KUKA KRL program: EPS_2_25716_MHDR06_A_20250926071555.src

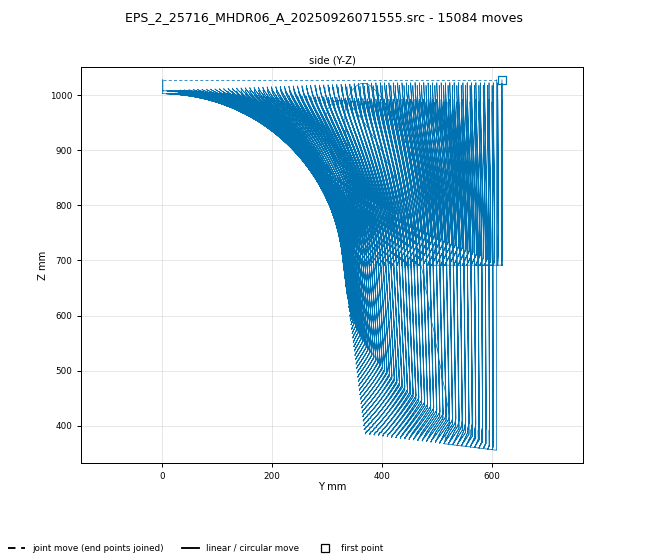
[picture p0: tool path of EPS_2_25716_MHDR06_A_20250926071555.src, 15084 of 15086 moves have a stored position in this frame; points joined in program order, loops and branches not executed]
&ACCESS RVP
&REL 4
&COMMENT QRS 19112012
&PARAM EDITMASK = *
DEF PART()
EXT BAS (BAS_COMMAND :IN,REAL :IN )
INT I
BAS (#INITMOV,0 )

;KUKA QRS Post kuka4.cps  Date:22-06-2017 !

File_ID=2855

QRS_PRE_INIT()

;Init var - Until changes are made in qrs_pre_init
Outlet_Square_prg=0
Inlet_1_Square_prg=0
Inlet_2_Square_prg=0
Inlet_3_Square_prg=0
Inlet_4_Square_prg=0
Inlet_5_Square_prg=0

Outlet_1={X 0.000, Y 400.000, Z 713.000, B 0.000, E1 0.000 }
Inlet_1={X 0.000, Y 400.000, Z 683.000, B 0.000, E1 180.000 }
Outlet_1_type=610
Inlet_1_type=610
;QRS#1=Sidecore dimensions
;QRS#2=600-24" Concrete
;QRS#3=600-24" Concrete
;QRS#4=
;QRS#5=
;QRS#6=
;QRS#7=
;QRS#8=
;QRS#9=S306-34L
;QRS#10=S306-34L
;QRS#11=
;QRS#12=
;QRS#13=
;QRS#14=
;QRS#15=
;QRS#16=1220x127x1372 4,5'
;QRS#17=EPS Height
;QRS#18=1018
;QRS#19=*
;QRS#20= UPDATED VERSION 22-06-2017
;QRS#21=*
Outlet_Square=0450
Inlet_1_Square=0450
Inlet_2_Square=0
Inlet_3_Square=0
Inlet_4_Square=0
Inlet_5_Square=0
Mill_Square=1
Outlet_Square_Prg=264
Inlet_1_Square_prg=264

QRS_INIT()

$ADVANCE=5

; T1
PTP {E1 171.02,E2 171.02}
PTP {X 0,Y 617.769,A -85,B 0,C 180,E1 171.02,E2 171.02,E3 0,E4 0,E5 0,E6 0}
QRS_SPEED_INIT()
LIN {X 0,Y 617.769,Z 1028,A -85,B 0,C 180,E1 171.02,E2 171.02,E3 0,E4 0,E5 0,E6 0} C_VEL
LIN {X 0,Y 617.769,Z 693.44,A -85,B 0,C 180,E1 171.02,E2 171.02} C_VEL
LIN {X 0,Y 617.8,Z 691.44,A -85,B 0,C 180,E1 171.206,E2 171.206} C_VEL
LIN {X 0,Y 617.968,Z 691.44,A -85,B 0,C 180,E1 171.885,E2 171.885} C_VEL
LIN {X 0,Y 618.013,Z 691.44,A -85,B 0,C 180,E1 176.532,E2 176.532} C_VEL
LIN {X 0,Y 618.047,Z 691.44,A -85,B 0,C 180,E1 181.155,E2 181.155} C_VEL
LIN {X 0,Y 617.982,Z 691.44,A -85,B 0,C 180,E1 185.787,E2 185.787} C_VEL
LIN {X 0,Y 617.952,Z 691.44,A -85,B 0,C 180,E1 190.457,E2 190.457} C_VEL
LIN {X 0,Y 617.972,Z 691.44,A -85,B 0,C 180,E1 195.197,E2 195.197} C_VEL
LIN {X 0,Y 617.907,Z 691.44,A -85,B 0,C 180,E1 200.05,E2 200.05} C_VEL
LIN {X 0,Y 617.438,Z 691.44,A -85,B 0,C 180,E1 202.548,E2 202.548} C_VEL
LIN {X 0,Y 617.908,Z 691.44,A -85,B 0,C 180,E1 205.056,E2 205.056} C_VEL
LIN {X 0,Y 617.398,Z 691.44,A -85,B 0,C 180,E1 207.66,E2 207.66} C_VEL
LIN {X 0,Y 617.843,Z 691.44,A -85,B 0,C 180,E1 210.28,E2 210.28} C_VEL
LIN {X 0,Y 617.317,Z 691.44,A -85,B 0,C 180,E1 213.027,E2 213.027} C_VEL
LIN {X 0,Y 617.82,Z 691.44,A -85,B 0,C 180,E1 215.798,E2 215.798} C_VEL
LIN {X 0,Y 617.574,Z 691.44,A -85,B 0,C 180,E1 218.108,E2 218.108} C_VEL
LIN {X 0,Y 617.547,Z 691.44,A -85,B 0,C 180,E1 218.722,E2 218.722} C_VEL
LIN {X 0,Y 617.751,Z 691.44,A -85,B 0,C 180,E1 221.735,E2 221.735} C_VEL
LIN {X 0,Y 617.856,Z 691.44,A -85,B 0,C 180,E1 225.104,E2 225.104} C_VEL
LIN {X 0,Y 617.438,Z 691.44,A -85,B 0,C 180,E1 228.31,E2 228.31} C_VEL
LIN {X 0,Y 617.785,Z 691.44,A -85,B 0,C 180,E1 231.301,E2 231.301} C_VEL
LIN {X 0,Y 617.972,Z 691.44,A -85,B 0,C 180,E1 236.345,E2 236.345} C_VEL
LIN {X 0,Y 617.889,Z 691.44,A -85,B 0,C 180,E1 236.677,E2 236.677} C_VEL
LIN {X 0,Y 617.182,Z 691.44,A -85,B 0,C 180,E1 236.802,E2 236.802} C_VEL
LIN {X 0,Y 616.593,Z 691.442,A -85,B 0,C 180,E1 236.859,E2 236.859} C_VEL
LIN {X 0,Y 617.379,Z 698.721,A -85,B 0,C 180,E1 237.005,E2 237.005} C_VEL
LIN {X 0,Y 617.562,Z 731.83,A -85,B 0,C 180,E1 237.472,E2 237.472} C_VEL
LIN {X 0,Y 617.518,Z 745.273,A -85,B 0,C 180,E1 237.692,E2 237.692} C_VEL
LIN {X 0,Y 617.627,Z 759.991,A -85,B 0,C 180,E1 238.015,E2 238.015} C_VEL
LIN {X 0,Y 617.596,Z 772.178,A -85,B 0,C 180,E1 238.333,E2 238.333} C_VEL
LIN {X 0,Y 617.775,Z 789.25,A -85,B 0,C 180,E1 238.876,E2 238.876} C_VEL
LIN {X 0,Y 617.661,Z 803.567,A -85,B 0,C 180,E1 239.398,E2 239.398} C_VEL
LIN {X 0,Y 617.795,Z 819.272,A -85,B 0,C 180,E1 240.077,E2 240.077} C_VEL
LIN {X 0,Y 617.796,Z 833.607,A -85,B 0,C 180,E1 240.772,E2 240.772} C_VEL
LIN {X 0,Y 617.742,Z 845.603,A -85,B 0,C 180,E1 241.41,E2 241.41} C_VEL
LIN {X 0,Y 617.842,Z 859.517,A -85,B 0,C 180,E1 242.243,E2 242.243} C_VEL
LIN {X 0,Y 617.838,Z 873.674,A -85,B 0,C 180,E1 243.177,E2 243.177} C_VEL
LIN {X 0,Y 617.828,Z 885.936,A -85,B 0,C 180,E1 244.063,E2 244.063} C_VEL
LIN {X 0,Y 617.821,Z 897.15,A -85,B 0,C 180,E1 244.943,E2 244.943} C_VEL
LIN {X 0,Y 617.854,Z 908.216,A -85,B 0,C 180,E1 245.886,E2 245.886} C_VEL
LIN {X 0,Y 617.903,Z 919.181,A -85,B 0,C 180,E1 246.901,E2 246.901} C_VEL
LIN {X 0,Y 617.832,Z 929.557,A -85,B 0,C 180,E1 247.938,E2 247.938} C_VEL
LIN {X 0,Y 617.851,Z 939.544,A -85,B 0,C 180,E1 249.026,E2 249.026} C_VEL
LIN {X 0,Y 617.957,Z 948.912,A -85,B 0,C 180,E1 250.137,E2 250.137} C_VEL
LIN {X 0,Y 617.805,Z 957.463,A -85,B 0,C 180,E1 251.226,E2 251.226} C_VEL
LIN {X 0,Y 617.797,Z 965.811,A -85,B 0,C 180,E1 252.391,E2 252.391} C_VEL
LIN {X 0,Y 617.997,Z 973.741,A -85,B 0,C 180,E1 253.613,E2 253.613} C_VEL
LIN {X 0,Y 617.808,Z 980.894,A -85,B 0,C 180,E1 254.801,E2 254.801} C_VEL
LIN {X 0,Y 617.811,Z 988.821,A -85,B 0,C 180,E1 256.292,E2 256.292} C_VEL
LIN {X 0,Y 617.963,Z 994.484,A -85,B 0,C 180,E1 257.482,E2 257.482} C_VEL
LIN {X 0,Y 617.732,Z 1000.738,A -85,B 0,C 180,E1 258.953,E2 258.953} C_VEL
LIN {X 0,Y 617.807,Z 1005.633,A -85,B 0,C 180,E1 260.289,E2 260.289} C_VEL
LIN {X 0,Y 617.976,Z 1008.324,A -85,B 0,C 180,E1 261.143,E2 261.143} C_VEL
LIN {X 0,Y 617.856,Z 1010.563,A -85,B 0,C 180,E1 261.885,E2 261.885} C_VEL
LIN {X 0,Y 617.743,Z 1013.111,A -85,B 0,C 180,E1 262.816,E2 262.816} C_VEL
LIN {X 0,Y 617.83,Z 1016.208,A -85,B 0,C 180,E1 264.213,E2 264.213} C_VEL
LIN {X 0,Y 617.976,Z 1017.804,A -85,B 0,C 180,E1 265.143,E2 265.143} C_VEL
LIN {X 0,Y 617.882,Z 1018.62,A -85,B 0,C 180,E1 265.605,E2 265.605} C_VEL
LIN {X 0,Y 617.751,Z 1019.844,A -85,B 0,C 180,E1 266.531,E2 266.531} C_VEL
LIN {X 0,Y 617.754,Z 1020.831,A -85,B 0,C 180,E1 267.457,E2 267.457} C_VEL
LIN {X 0,Y 617.996,Z 1021.643,A -85,B 0,C 180,E1 268.845,E2 268.845} C_VEL
LIN {X 0,Y 617.666,Z 1021.732,A -85,B 0,C 180,E1 271.156,E2 271.156} C_VEL
LIN {X 0,Y 617.88,Z 1020.797,A -85,B 0,C 180,E1 272.543,E2 272.543} C_VEL
LIN {X 0,Y 617.842,Z 1019.819,A -85,B 0,C 180,E1 273.469,E2 273.469} C_VEL
LIN {X 0,Y 617.732,Z 1018.658,A -85,B 0,C 180,E1 274.396,E2 274.396} C_VEL
LIN {X 0,Y 617.804,Z 1016.213,A -85,B 0,C 180,E1 275.788,E2 275.788} C_VEL
LIN {X 0,Y 617.988,Z 1014.126,A -85,B 0,C 180,E1 276.716,E2 276.716} C_VEL
LIN {X 0,Y 617.83,Z 1011.822,A -85,B 0,C 180,E1 277.649,E2 277.649} C_VEL
LIN {X 0,Y 617.78,Z 1008.462,A -85,B 0,C 180,E1 278.832,E2 278.832} C_VEL
LIN {X 0,Y 617.963,Z 1004.405,A -85,B 0,C 180,E1 280.048,E2 280.048} C_VEL
LIN {X 0,Y 617.795,Z 999.566,A -85,B 0,C 180,E1 281.341,E2 281.341} C_VEL
LIN {X 0,Y 617.74,Z 994.527,A -85,B 0,C 180,E1 282.523,E2 282.523} C_VEL
LIN {X 0,Y 617.975,Z 987.305,A -85,B 0,C 180,E1 284.002,E2 284.002} C_VEL
LIN {X 0,Y 617.805,Z 979.862,A -85,B 0,C 180,E1 285.374,E2 285.374} C_VEL
LIN {X 0,Y 617.795,Z 972.028,A -85,B 0,C 180,E1 286.666,E2 286.666} C_VEL
LIN {X 0,Y 617.958,Z 964.032,A -85,B 0,C 180,E1 287.857,E2 287.857} C_VEL
LIN {X 0,Y 617.819,Z 955.95,A -85,B 0,C 180,E1 288.977,E2 288.977} C_VEL
LIN {X 0,Y 617.839,Z 946.158,A -85,B 0,C 180,E1 290.204,E2 290.204} C_VEL
LIN {X 0,Y 617.952,Z 936.782,A -85,B 0,C 180,E1 291.281,E2 291.281} C_VEL
LIN {X 0,Y 617.847,Z 926.511,A -85,B 0,C 180,E1 292.374,E2 292.374} C_VEL
LIN {X 0,Y 617.845,Z 916.724,A -85,B 0,C 180,E1 293.335,E2 293.335} C_VEL
LIN {X 0,Y 617.862,Z 905.186,A -85,B 0,C 180,E1 294.376,E2 294.376} C_VEL
LIN {X 0,Y 617.853,Z 894.173,A -85,B 0,C 180,E1 295.295,E2 295.295} C_VEL
LIN {X 0,Y 617.838,Z 881.592,A -85,B 0,C 180,E1 296.259,E2 296.259} C_VEL
LIN {X 0,Y 617.824,Z 870.134,A -85,B 0,C 180,E1 297.067,E2 297.067} C_VEL
LIN {X 0,Y 617.85,Z 856.712,A -85,B 0,C 180,E1 297.928,E2 297.928} C_VEL
LIN {X 0,Y 617.812,Z 842.841,A -85,B 0,C 180,E1 298.735,E2 298.735} C_VEL
LIN {X 0,Y 617.728,Z 831.67,A -85,B 0,C 180,E1 299.334,E2 299.334} C_VEL
LIN {X 0,Y 617.799,Z 815.203,A -85,B 0,C 180,E1 300.103,E2 300.103} C_VEL
LIN {X 0,Y 617.676,Z 801.179,A -85,B 0,C 180,E1 300.691,E2 300.691} C_VEL
LIN {X 0,Y 617.671,Z 792.906,A -85,B 0,C 180,E1 300.996,E2 300.996} C_VEL
LIN {X 0,Y 617.767,Z 783.913,A -85,B 0,C 180,E1 301.296,E2 301.296} C_VEL
LIN {X 0,Y 617.782,Z 774.18,A -85,B 0,C 180,E1 301.602,E2 301.602} C_VEL
LIN {X 0,Y 617.522,Z 758.624,A -85,B 0,C 180,E1 302.025,E2 302.025} C_VEL
LIN {X 0,Y 617.763,Z 743.298,A -85,B 0,C 180,E1 302.332,E2 302.332} C_VEL
LIN {X 0,Y 617.696,Z 723.174,A -85,B 0,C 180,E1 302.644,E2 302.644} C_VEL
LIN {X 0,Y 617.36,Z 698.518,A -85,B 0,C 180,E1 302.998,E2 302.998} C_VEL
LIN {X 0,Y 616.602,Z 691.44,A -85,B 0,C 180,E1 303.143,E2 303.143} C_VEL
LIN {X 0,Y 617.104,Z 691.44,A -85,B 0,C 180,E1 303.189,E2 303.189} C_VEL
LIN {X 0,Y 617.789,Z 691.44,A -85,B 0,C 180,E1 303.3,E2 303.3} C_VEL
LIN {X 0,Y 618.014,Z 691.44,A -85,B 0,C 180,E1 303.592,E2 303.592} C_VEL
LIN {X 0,Y 617.789,Z 691.44,A -85,B 0,C 180,E1 308.699,E2 308.699} C_VEL
LIN {X 0,Y 617.439,Z 691.44,A -85,B 0,C 180,E1 311.755,E2 311.755} C_VEL
LIN {X 0,Y 617.857,Z 691.44,A -85,B 0,C 180,E1 314.897,E2 314.897} C_VEL
LIN {X 0,Y 617.756,Z 691.44,A -85,B 0,C 180,E1 318.27,E2 318.27} C_VEL
LIN {X 0,Y 617.543,Z 691.44,A -85,B 0,C 180,E1 321.278,E2 321.278} C_VEL
LIN {X 0,Y 617.577,Z 691.44,A -85,B 0,C 180,E1 321.893,E2 321.893} C_VEL
LIN {X 0,Y 617.818,Z 691.44,A -85,B 0,C 180,E1 324.202,E2 324.202} C_VEL
LIN {X 0,Y 617.322,Z 691.44,A -85,B 0,C 180,E1 326.974,E2 326.974} C_VEL
LIN {X 0,Y 617.835,Z 691.44,A -85,B 0,C 180,E1 329.719,E2 329.719} C_VEL
LIN {X 0,Y 617.381,Z 691.44,A -85,B 0,C 180,E1 332.339,E2 332.339} C_VEL
LIN {X 0,Y 617.882,Z 691.44,A -85,B 0,C 180,E1 334.943,E2 334.943} C_VEL
LIN {X 0,Y 617.416,Z 691.44,A -85,B 0,C 180,E1 337.451,E2 337.451} C_VEL
LIN {X 0,Y 617.909,Z 691.44,A -85,B 0,C 180,E1 339.95,E2 339.95} C_VEL
LIN {X 0,Y 617.993,Z 691.44,A -85,B 0,C 180,E1 343.627,E2 343.627} C_VEL
LIN {X 0,Y 617.927,Z 691.44,A -85,B 0,C 180,E1 349.543,E2 349.543} C_VEL
LIN {X 0,Y 617.984,Z 691.44,A -85,B 0,C 180,E1 354.213,E2 354.213} C_VEL
LIN {X 0,Y 618.053,Z 691.44,A -85,B 0,C 180,E1 358.845,E2 358.845} C_VEL
LIN {X 0,Y 618.006,Z 691.44,A -85,B 0,C 180,E1 363.468,E2 363.468} C_VEL
LIN {X 0,Y 617.974,Z 691.44,A -85,B 0,C 180,E1 368.115,E2 368.115} C_VEL
LIN {X 0,Y 617.996,Z 691.44,A -85,B 0,C 180,E1 372.815,E2 372.815} C_VEL
LIN {X 0,Y 617.957,Z 691.44,A -85,B 0,C 180,E1 377.607,E2 377.607} C_VEL
LIN {X 0,Y 617.756,Z 691.44,A -85,B 0,C 180,E1 378.561,E2 378.561} C_VEL
LIN {X 0,Y 617.91,Z 691.44,A -85,B 0,C 180,E1 382.53,E2 382.53} C_VEL
LIN {X 0,Y 617.424,Z 691.44,A -85,B 0,C 180,E1 385.077,E2 385.077} C_VEL
LIN {X 0,Y 617.883,Z 691.44,A -85,B 0,C 180,E1 387.637,E2 387.637} C_VEL
LIN {X 0,Y 617.432,Z 691.44,A -85,B 0,C 180,E1 390.302,E2 390.302} C_VEL
LIN {X 0,Y 617.966,Z 691.44,A -85,B 0,C 180,E1 392.988,E2 392.988} C_VEL
LIN {X 0,Y 617.693,Z 691.44,A -85,B 0,C 180,E1 395.806,E2 395.806} C_VEL
LIN {X 0,Y 617.694,Z 691.44,A -85,B 0,C 180,E1 398.121,E2 398.121} C_VEL
LIN {X 0,Y 617.812,Z 691.44,A -85,B 0,C 180,E1 401.736,E2 401.736} C_VEL
LIN {X 0,Y 617.415,Z 691.44,A -85,B 0,C 180,E1 405.062,E2 405.062} C_VEL
LIN {X 0,Y 617.817,Z 691.44,A -85,B 0,C 180,E1 408.276,E2 408.276} C_VEL
LIN {X 0,Y 617.727,Z 691.44,A -85,B 0,C 180,E1 411.882,E2 411.882} C_VEL
LIN {X 0,Y 617.729,Z 691.44,A -85,B 0,C 180,E1 414.2,E2 414.2} C_VEL
LIN {X 0,Y 617.795,Z 691.44,A -85,B 0,C 180,E1 415.792,E2 415.792} C_VEL
LIN {X 0,Y 617.754,Z 691.44,A -85,B 0,C 180,E1 417.003,E2 417.003} C_VEL
LIN {X 0,Y 617.547,Z 700.565,A -85,B 0,C 180,E1 417.406,E2 417.406} C_VEL
LIN {X 0,Y 617.667,Z 715.154,A -85,B 0,C 180,E1 417.653,E2 417.653} C_VEL
LIN {X 0,Y 617.521,Z 730.803,A -85,B 0,C 180,E1 417.985,E2 417.985} C_VEL
LIN {X 0,Y 617.762,Z 746.117,A -85,B 0,C 180,E1 418.413,E2 418.413} C_VEL
LIN {X 0,Y 617.721,Z 761.16,A -85,B 0,C 180,E1 418.898,E2 418.898} C_VEL
LIN {X 0,Y 617.647,Z 771.287,A -85,B 0,C 180,E1 419.267,E2 419.267} C_VEL
LIN {X 0,Y 617.812,Z 788.844,A -85,B 0,C 180,E1 420.012,E2 420.012} C_VEL
LIN {X 0,Y 617.71,Z 803.562,A -85,B 0,C 180,E1 420.72,E2 420.72} C_VEL
LIN {X 0,Y 617.82,Z 816.37,A -85,B 0,C 180,E1 421.414,E2 421.414} C_VEL
LIN {X 0,Y 617.848,Z 830.932,A -85,B 0,C 180,E1 422.29,E2 422.29} C_VEL
LIN {X 0,Y 617.783,Z 843.16,A -85,B 0,C 180,E1 423.093,E2 423.093} C_VEL
LIN {X 0,Y 617.824,Z 855.473,A -85,B 0,C 180,E1 423.982,E2 423.982} C_VEL
LIN {X 0,Y 617.846,Z 867.672,A -85,B 0,C 180,E1 424.944,E2 424.944} C_VEL
LIN {X 0,Y 617.863,Z 878.611,A -85,B 0,C 180,E1 425.878,E2 425.878} C_VEL
LIN {X 0,Y 617.83,Z 889.973,A -85,B 0,C 180,E1 426.932,E2 426.932} C_VEL
LIN {X 0,Y 617.877,Z 899.967,A -85,B 0,C 180,E1 427.939,E2 427.939} C_VEL
LIN {X 0,Y 617.955,Z 908.593,A -85,B 0,C 180,E1 428.874,E2 428.874} C_VEL
LIN {X 0,Y 617.815,Z 919.245,A -85,B 0,C 180,E1 430.128,E2 430.128} C_VEL
LIN {X 0,Y 617.837,Z 927.602,A -85,B 0,C 180,E1 431.202,E2 431.202} C_VEL
LIN {X 0,Y 617.942,Z 936.082,A -85,B 0,C 180,E1 432.394,E2 432.394} C_VEL
LIN {X 0,Y 617.763,Z 944.459,A -85,B 0,C 180,E1 433.676,E2 433.676} C_VEL
LIN {X 0,Y 617.824,Z 951.132,A -85,B 0,C 180,E1 434.8,E2 434.8} C_VEL
LIN {X 0,Y 617.979,Z 957.548,A -85,B 0,C 180,E1 435.998,E2 435.998} C_VEL
LIN {X 0,Y 617.736,Z 964.719,A -85,B 0,C 180,E1 437.477,E2 437.477} C_VEL
LIN {X 0,Y 617.804,Z 969.758,A -85,B 0,C 180,E1 438.659,E2 438.659} C_VEL
LIN {X 0,Y 617.968,Z 974.595,A -85,B 0,C 180,E1 439.958,E2 439.958} C_VEL
LIN {X 0,Y 617.756,Z 978.96,A -85,B 0,C 180,E1 441.275,E2 441.275} C_VEL
LIN {X 0,Y 617.845,Z 983.206,A -85,B 0,C 180,E1 442.817,E2 442.817} C_VEL
LIN {X 0,Y 617.962,Z 985.246,A -85,B 0,C 180,E1 443.749,E2 443.749} C_VEL
LIN {X 0,Y 617.792,Z 987.146,A -85,B 0,C 180,E1 444.676,E2 444.676} C_VEL
LIN {X 0,Y 617.736,Z 988.734,A -85,B 0,C 180,E1 445.604,E2 445.604} C_VEL
LIN {X 0,Y 617.822,Z 989.878,A -85,B 0,C 180,E1 446.531,E2 446.531} C_VEL
LIN {X 0,Y 617.972,Z 990.803,A -85,B 0,C 180,E1 447.457,E2 447.457} C_VEL
LIN {X 0,Y 617.716,Z 991.728,A -85,B 0,C 180,E1 448.844,E2 448.844} C_VEL
LIN {X 0,Y 617.923,Z 991.653,A -85,B 0,C 180,E1 451.155,E2 451.155} C_VEL
LIN {X 0,Y 617.765,Z 990.797,A -85,B 0,C 180,E1 452.543,E2 452.543} C_VEL
LIN {X 0,Y 617.677,Z 989.809,A -85,B 0,C 180,E1 453.469,E2 453.469} C_VEL
LIN {X 0,Y 617.742,Z 988.579,A -85,B 0,C 180,E1 454.396,E2 454.396} C_VEL
LIN {X 0,Y 617.919,Z 986.085,A -85,B 0,C 180,E1 455.786,E2 455.786} C_VEL
LIN {X 0,Y 617.727,Z 982.992,A -85,B 0,C 180,E1 457.184,E2 457.184} C_VEL
LIN {X 0,Y 617.798,Z 979.363,A -85,B 0,C 180,E1 458.507,E2 458.507} C_VEL
LIN {X 0,Y 617.934,Z 975.572,A -85,B 0,C 180,E1 459.674,E2 459.674} C_VEL
LIN {X 0,Y 617.754,Z 969.384,A -85,B 0,C 180,E1 461.341,E2 461.341} C_VEL
LIN {X 0,Y 617.889,Z 964.306,A -85,B 0,C 180,E1 462.52,E2 462.52} C_VEL
LIN {X 0,Y 617.89,Z 960.018,A -85,B 0,C 180,E1 463.409,E2 463.409} C_VEL
LIN {X 0,Y 617.758,Z 955.491,A -85,B 0,C 180,E1 464.304,E2 464.304} C_VEL
LIN {X 0,Y 617.765,Z 949.526,A -85,B 0,C 180,E1 465.387,E2 465.387} C_VEL
LIN {X 0,Y 617.977,Z 942.352,A -85,B 0,C 180,E1 466.563,E2 466.563} C_VEL
LIN {X 0,Y 617.805,Z 933.783,A -85,B 0,C 180,E1 467.854,E2 467.854} C_VEL
LIN {X 0,Y 617.794,Z 925.779,A -85,B 0,C 180,E1 468.954,E2 468.954} C_VEL
LIN {X 0,Y 617.962,Z 915.769,A -85,B 0,C 180,E1 470.199,E2 470.199} C_VEL
LIN {X 0,Y 617.846,Z 906.373,A -85,B 0,C 180,E1 471.284,E2 471.284} C_VEL
LIN {X 0,Y 617.826,Z 896.063,A -85,B 0,C 180,E1 472.374,E2 472.374} C_VEL
LIN {X 0,Y 617.902,Z 886.089,A -85,B 0,C 180,E1 473.345,E2 473.345} C_VEL
LIN {X 0,Y 617.877,Z 876.237,A -85,B 0,C 180,E1 474.242,E2 474.242} C_VEL
LIN {X 0,Y 617.845,Z 863.602,A -85,B 0,C 180,E1 475.295,E2 475.295} C_VEL
LIN {X 0,Y 617.816,Z 852.103,A -85,B 0,C 180,E1 476.178,E2 476.178} C_VEL
LIN {X 0,Y 617.858,Z 839.452,A -85,B 0,C 180,E1 477.065,E2 477.065} C_VEL
LIN {X 0,Y 617.837,Z 826.763,A -85,B 0,C 180,E1 477.88,E2 477.88} C_VEL
LIN {X 0,Y 617.724,Z 813.694,A -85,B 0,C 180,E1 478.649,E2 478.649} C_VEL
LIN {X 0,Y 617.815,Z 799.775,A -85,B 0,C 180,E1 479.376,E2 479.376} C_VEL
LIN {X 0,Y 617.769,Z 785.259,A -85,B 0,C 180,E1 480.058,E2 480.058} C_VEL
LIN {X 0,Y 617.652,Z 771.869,A -85,B 0,C 180,E1 480.622,E2 480.622} C_VEL
LIN {X 0,Y 617.768,Z 756.723,A -85,B 0,C 180,E1 481.162,E2 481.162} C_VEL
LIN {X 0,Y 617.634,Z 741.567,A -85,B 0,C 180,E1 481.635,E2 481.635} C_VEL
LIN {X 0,Y 617.622,Z 734.394,A -85,B 0,C 180,E1 481.825,E2 481.825} C_VEL
LIN {X 0,Y 617.755,Z 725.284,A -85,B 0,C 180,E1 482.038,E2 482.038} C_VEL
LIN {X 0,Y 617.77,Z 711.173,A -85,B 0,C 180,E1 482.321,E2 482.321} C_VEL
LIN {X 0,Y 617.397,Z 692.323,A -85,B 0,C 180,E1 482.628,E2 482.628} C_VEL
LIN {X 0,Y 617.467,Z 691.44,A -85,B 0,C 180,E1 482.656,E2 482.656} C_VEL
LIN {X 0,Y 618.076,Z 691.44,A -85,B 0,C 180,E1 482.977,E2 482.977} C_VEL
LIN {X 0,Y 617.727,Z 691.44,A -85,B 0,C 180,E1 484.199,E2 484.199} C_VEL
LIN {X 0,Y 617.784,Z 691.44,A -85,B 0,C 180,E1 488.699,E2 488.699} C_VEL
LIN {X 0,Y 617.435,Z 691.44,A -85,B 0,C 180,E1 491.755,E2 491.755} C_VEL
LIN {X 0,Y 617.864,Z 691.44,A -85,B 0,C 180,E1 494.895,E2 494.895} C_VEL
LIN {X 0,Y 617.761,Z 691.44,A -85,B 0,C 180,E1 498.268,E2 498.268} C_VEL
LIN {X 0,Y 617.553,Z 691.44,A -85,B 0,C 180,E1 501.278,E2 501.278} C_VEL
LIN {X 0,Y 617.828,Z 691.44,A -85,B 0,C 180,E1 504.203,E2 504.203} C_VEL
LIN {X 0,Y 617.326,Z 691.44,A -85,B 0,C 180,E1 506.974,E2 506.974} C_VEL
LIN {X 0,Y 617.855,Z 691.44,A -85,B 0,C 180,E1 509.72,E2 509.72} C_VEL
LIN {X 0,Y 617.415,Z 691.44,A -85,B 0,C 180,E1 512.341,E2 512.341} C_VEL
LIN {X 0,Y 617.927,Z 691.44,A -85,B 0,C 180,E1 514.945,E2 514.945} C_VEL
LIN {X 0,Y 617.447,Z 691.44,A -85,B 0,C 180,E1 517.452,E2 517.452} C_VEL
LIN {X 0,Y 617.926,Z 691.44,A -85,B 0,C 180,E1 519.951,E2 519.951} C_VEL
LIN {X 0,Y 617.695,Z 691.44,A -85,B 0,C 180,E1 522.386,E2 522.386} C_VEL
LIN {X 0,Y 617.79,Z 691.44,A -85,B 0,C 180,E1 524.798,E2 524.798} C_VEL
LIN {X 0,Y 617.994,Z 691.44,A -85,B 0,C 180,E1 527.185,E2 527.185} C_VEL
LIN {X 0,Y 617.8,Z 691.44,A -85,B 0,C 180,E1 531.206,E2 531.206} C_VEL
LIN {X 0,Y 615.264,Z 691.44,A -85,B 0,C 180,E1 532.402,E2 532.402} C_VEL
LIN {X 0,Y 609.688,Z 691.44,A -85,B 0,C 180,E1 534.19,E2 534.19} C_VEL
LIN {X 0,Y 609.601,Z 691.44,A -85,B 0,C 180,E1 534.397,E2 534.397} C_VEL
LIN {X 0,Y 609.633,Z 691.44,A -85,B 0,C 180,E1 538.58,E2 538.58} C_VEL
LIN {X 0,Y 609.667,Z 691.44,A -85,B 0,C 180,E1 542.85,E2 542.85} C_VEL
LIN {X 0,Y 609.66,Z 691.44,A -85,B 0,C 180,E1 547.136,E2 547.136} C_VEL
LIN {X 0,Y 609.73,Z 691.44,A -85,B 0,C 180,E1 551.46,E2 551.46} C_VEL
LIN {X 0,Y 609.801,Z 691.44,A -85,B 0,C 180,E1 555.851,E2 555.851} C_VEL
LIN {X 0,Y 609.92,Z 691.44,A -85,B 0,C 180,E1 560.338,E2 560.338} C_VEL
LIN {X 0,Y 609.993,Z 691.44,A -85,B 0,C 180,E1 564.959,E2 564.959} C_VEL
LIN {X 0,Y 609.763,Z 691.44,A -85,B 0,C 180,E1 569.776,E2 569.776} C_VEL
LIN {X 0,Y 609.756,Z 691.44,A -85,B 0,C 180,E1 576.578,E2 576.578} C_VEL
LIN {X 0,Y 609.76,Z 691.44,A -85,B 0,C 180,E1 582.098,E2 582.098} C_VEL
LIN {X 0,Y 609.482,Z 691.44,A -85,B 0,C 180,E1 587.876,E2 587.876} C_VEL
LIN {X 0,Y 609.483,Z 691.44,A -85,B 0,C 180,E1 592.645,E2 592.645} C_VEL
LIN {X 0,Y 610.01,Z 691.44,A -85,B 0,C 180,E1 596.454,E2 596.454} C_VEL
LIN {X 0,Y 610.899,Z 757.873,A -85,B 0,C 180,E1 597.569,E2 597.569} C_VEL
LIN {X 0,Y 610.811,Z 798.846,A -85,B 0,C 180,E1 598.839,E2 598.839} C_VEL
LIN {X 0,Y 610.68,Z 836.968,A -85,B 0,C 180,E1 600.58,E2 600.58} C_VEL
LIN {X 0,Y 610.553,Z 873.915,A -85,B 0,C 180,E1 602.848,E2 602.848} C_VEL
LIN {X 0,Y 610.356,Z 909.006,A -85,B 0,C 180,E1 605.645,E2 605.645} C_VEL
LIN {X 0,Y 610.19,Z 940.958,A -85,B 0,C 180,E1 608.913,E2 608.913} C_VEL
LIN {X 0,Y 610.055,Z 966.925,A -85,B 0,C 180,E1 612.3,E2 612.3} C_VEL
LIN {X 0,Y 610.009,Z 988.719,A -85,B 0,C 180,E1 615.996,E2 615.996} C_VEL
LIN {X 0,Y 609.944,Z 1004.432,A -85,B 0,C 180,E1 619.632,E2 619.632} C_VEL
LIN {X 0,Y 609.925,Z 1014.987,A -85,B 0,C 180,E1 623.161,E2 623.161} C_VEL
LIN {X 0,Y 610.059,Z 1019.905,A -85,B 0,C 180,E1 625.73,E2 625.73} C_VEL
LIN {X 0,Y 610.113,Z 1022.657,A -85,B 0,C 180,E1 628.578,E2 628.578} C_VEL
LIN {X 0,Y 610.063,Z 1021.627,A -85,B 0,C 180,E1 632.845,E2 632.845} C_VEL
LIN {X 0,Y 610.093,Z 1014.331,A -85,B 0,C 180,E1 637.128,E2 637.128} C_VEL
LIN {X 0,Y 610,Z 1001.733,A -85,B 0,C 180,E1 641.091,E2 641.091} C_VEL
LIN {X 0,Y 610.062,Z 984.702,A -85,B 0,C 180,E1 644.755,E2 644.755} C_VEL
LIN {X 0,Y 610.17,Z 963.033,A -85,B 0,C 180,E1 648.257,E2 648.257} C_VEL
LIN {X 0,Y 610.292,Z 935.926,A -85,B 0,C 180,E1 651.656,E2 651.656} C_VEL
LIN {X 0,Y 610.394,Z 903.442,A -85,B 0,C 180,E1 654.843,E2 654.843} C_VEL
LIN {X 0,Y 610.558,Z 868.357,A -85,B 0,C 180,E1 657.534,E2 657.534} C_VEL
LIN {X 0,Y 610.703,Z 829.52,A -85,B 0,C 180,E1 659.81,E2 659.81} C_VEL
LIN {X 0,Y 610.937,Z 789.147,A -85,B 0,C 180,E1 661.516,E2 661.516} C_VEL
LIN {X 0,Y 610.984,Z 749.991,A -85,B 0,C 180,E1 662.595,E2 662.595} C_VEL
LIN {X 0,Y 610.011,Z 691.44,A -85,B 0,C 180,E1 663.547,E2 663.547} C_VEL
LIN {X 0,Y 609.591,Z 691.44,A -85,B 0,C 180,E1 669.653,E2 669.653} C_VEL
LIN {X 0,Y 609.712,Z 691.44,A -85,B 0,C 180,E1 675.95,E2 675.95} C_VEL
LIN {X 0,Y 609.547,Z 691.44,A -85,B 0,C 180,E1 680.357,E2 680.357} C_VEL
LIN {X 0,Y 609.603,Z 691.44,A -85,B 0,C 180,E1 685.164,E2 685.164} C_VEL
LIN {X 0,Y 609.716,Z 691.44,A -85,B 0,C 180,E1 690.36,E2 690.36} C_VEL
LIN {X 0,Y 609.958,Z 691.44,A -85,B 0,C 180,E1 695.04,E2 695.04} C_VEL
LIN {X 0,Y 609.758,Z 691.44,A -85,B 0,C 180,E1 701.167,E2 701.167} C_VEL
LIN {X 0,Y 609.344,Z 691.44,A -85,B 0,C 180,E1 705.611,E2 705.611} C_VEL
LIN {X 0,Y 609.867,Z 691.44,A -85,B 0,C 180,E1 709.99,E2 709.99} C_VEL
LIN {X 0,Y 610.066,Z 691.44,A -85,B 0,C 180,E1 714.3,E2 714.3} C_VEL
LIN {X 0,Y 609.769,Z 691.44,A -85,B 0,C 180,E1 719.997,E2 719.997} C_VEL
LIN {X 0,Y 609.809,Z 691.44,A -85,B 0,C 180,E1 724.268,E2 724.268} C_VEL
LIN {X 0,Y 609.913,Z 691.44,A -85,B 0,C 180,E1 728.561,E2 728.561} C_VEL
LIN {X 0,Y 610.051,Z 691.44,A -85,B 0,C 180,E1 732.902,E2 732.902} C_VEL
LIN {X 0,Y 609.779,Z 691.44,A -85,B 0,C 180,E1 738.825,E2 738.825} C_VEL
LIN {X 0,Y 609.735,Z 691.44,A -85,B 0,C 180,E1 743.403,E2 743.403} C_VEL
LIN {X 0,Y 609.802,Z 691.44,A -85,B 0,C 180,E1 748.14,E2 748.14} C_VEL
LIN {X 0,Y 610.028,Z 691.44,A -85,B 0,C 180,E1 753.086,E2 753.086} C_VEL
LIN {X 0,Y 609.735,Z 691.44,A -85,B 0,C 180,E1 758.364,E2 758.364} C_VEL
LIN {X 0,Y 609.775,Z 691.44,A -85,B 0,C 180,E1 762.087,E2 762.087} C_VEL
LIN {X 0,Y 609.857,Z 691.44,A -85,B 0,C 180,E1 768.128,E2 768.128} C_VEL
LIN {X 0,Y 609.735,Z 691.44,A -85,B 0,C 180,E1 773.418,E2 773.418} C_VEL
LIN {X 0,Y 609.852,Z 691.44,A -85,B 0,C 180,E1 776.787,E2 776.787} C_VEL
LIN {X 0,Y 610.888,Z 724.267,A -85,B 0,C 180,E1 777.446,E2 777.446} C_VEL
LIN {X 0,Y 610.819,Z 764.473,A -85,B 0,C 180,E1 778.631,E2 778.631} C_VEL
LIN {X 0,Y 610.645,Z 804.023,A -85,B 0,C 180,E1 780.373,E2 780.373} C_VEL
LIN {X 0,Y 610.52,Z 842.903,A -85,B 0,C 180,E1 782.728,E2 782.728} C_VEL
LIN {X 0,Y 610.352,Z 878.953,A -85,B 0,C 180,E1 785.594,E2 785.594} C_VEL
LIN {X 0,Y 610.282,Z 909.722,A -85,B 0,C 180,E1 788.725,E2 788.725} C_VEL
LIN {X 0,Y 610.207,Z 937.215,A -85,B 0,C 180,E1 792.304,E2 792.304} C_VEL
LIN {X 0,Y 610.163,Z 958.934,A -85,B 0,C 180,E1 795.999,E2 795.999} C_VEL
LIN {X 0,Y 610.165,Z 975.945,A -85,B 0,C 180,E1 799.997,E2 799.997} C_VEL
LIN {X 0,Y 610.04,Z 987.566,A -85,B 0,C 180,E1 804.302,E2 804.302} C_VEL
LIN {X 0,Y 610.094,Z 991.671,A -85,B 0,C 180,E1 807.155,E2 807.155} C_VEL
LIN {X 0,Y 610.047,Z 992.628,A -85,B 0,C 180,E1 811.422,E2 811.422} C_VEL
LIN {X 0,Y 610.093,Z 987.383,A -85,B 0,C 180,E1 815.697,E2 815.697} C_VEL
LIN {X 0,Y 610.072,Z 975.612,A -85,B 0,C 180,E1 820.004,E2 820.004} C_VEL
LIN {X 0,Y 610.015,Z 958.492,A -85,B 0,C 180,E1 824.004,E2 824.004} C_VEL
LIN {X 0,Y 610.089,Z 935.393,A -85,B 0,C 180,E1 827.885,E2 827.885} C_VEL
LIN {X 0,Y 610.192,Z 907.277,A -85,B 0,C 180,E1 831.469,E2 831.469} C_VEL
LIN {X 0,Y 610.379,Z 875.213,A -85,B 0,C 180,E1 834.648,E2 834.648} C_VEL
LIN {X 0,Y 610.589,Z 839.027,A -85,B 0,C 180,E1 837.443,E2 837.443} C_VEL
LIN {X 0,Y 610.764,Z 800.347,A -85,B 0,C 180,E1 839.722,E2 839.722} C_VEL
LIN {X 0,Y 610.908,Z 760.558,A -85,B 0,C 180,E1 841.42,E2 841.42} C_VEL
LIN {X 0,Y 611.049,Z 723.164,A -85,B 0,C 180,E1 842.478,E2 842.478} C_VEL
LIN {X 0,Y 610.149,Z 691.44,A -85,B 0,C 180,E1 843.088,E2 843.088} C_VEL
LIN {X 0,Y 609.597,Z 691.44,A -85,B 0,C 180,E1 849.665,E2 849.665} C_VEL
LIN {X 0,Y 609.706,Z 691.44,A -85,B 0,C 180,E1 855.959,E2 855.959} C_VEL
LIN {X 0,Y 609.537,Z 691.44,A -85,B 0,C 180,E1 860.357,E2 860.357} C_VEL
LIN {X 0,Y 609.602,Z 691.44,A -85,B 0,C 180,E1 865.172,E2 865.172} C_VEL
LIN {X 0,Y 609.737,Z 691.44,A -85,B 0,C 180,E1 870.355,E2 870.355} C_VEL
LIN {X 0,Y 610.007,Z 691.44,A -85,B 0,C 180,E1 875.05,E2 875.05} C_VEL
LIN {X 0,Y 609.8,Z 691.44,A -85,B 0,C 180,E1 881.175,E2 881.175} C_VEL
LIN {X 0,Y 610.082,Z 691.44,A -85,B 0,C 180,E1 887.099,E2 887.099} C_VEL
LIN {X 0,Y 609.747,Z 691.44,A -85,B 0,C 180,E1 892.872,E2 892.872} C_VEL
LIN {X 0,Y 609.601,Z 691.44,A -85,B 0,C 180,E1 894.397,E2 894.397} C_VEL
LIN {X 0,Y 605.848,Z 691.44,A -85,B 0,C 180,E1 896.004,E2 896.004} C_VEL
LIN {X 0,Y 601.857,Z 691.44,A -85,B 0,C 180,E1 897.631,E2 897.631} C_VEL
LIN {X 0,Y 602.139,Z 691.44,A -85,B 0,C 180,E1 901.444,E2 901.444} C_VEL
LIN {X 0,Y 602.138,Z 691.44,A -85,B 0,C 180,E1 905.775,E2 905.775} C_VEL
LIN {X 0,Y 601.818,Z 691.44,A -85,B 0,C 180,E1 911.613,E2 911.613} C_VEL
LIN {X 0,Y 601.831,Z 691.44,A -85,B 0,C 180,E1 916.067,E2 916.067} C_VEL
LIN {X 0,Y 601.722,Z 691.44,A -85,B 0,C 180,E1 921.407,E2 921.407} C_VEL
LIN {X 0,Y 601.971,Z 691.44,A -85,B 0,C 180,E1 925.315,E2 925.315} C_VEL
LIN {X 0,Y 601.68,Z 691.44,A -85,B 0,C 180,E1 931.176,E2 931.176} C_VEL
LIN {X 0,Y 601.776,Z 691.44,A -85,B 0,C 180,E1 937.144,E2 937.144} C_VEL
LIN {X 0,Y 601.75,Z 691.44,A -85,B 0,C 180,E1 943.141,E2 943.141} C_VEL
LIN {X 0,Y 601.56,Z 691.44,A -85,B 0,C 180,E1 949.126,E2 949.126} C_VEL
LIN {X 0,Y 601.495,Z 691.44,A -85,B 0,C 180,E1 953.654,E2 953.654} C_VEL
LIN {X 0,Y 601.973,Z 691.44,A -85,B 0,C 180,E1 955.945,E2 955.945} C_VEL
LIN {X 0,Y 604.134,Z 701.027,A -85,B 0,C 180,E1 956.218,E2 956.218} C_VEL
LIN {X 0,Y 604.213,Z 757.523,A -85,B 0,C 180,E1 957.158,E2 957.158} C_VEL
LIN {X 0,Y 603.981,Z 798.327,A -85,B 0,C 180,E1 958.427,E2 958.427} C_VEL
LIN {X 0,Y 603.612,Z 837.137,A -85,B 0,C 180,E1 960.21,E2 960.21} C_VEL
LIN {X 0,Y 603.28,Z 873.611,A -85,B 0,C 180,E1 962.471,E2 962.471} C_VEL
LIN {X 0,Y 602.864,Z 909,A -85,B 0,C 180,E1 965.321,E2 965.321} C_VEL
LIN {X 0,Y 602.517,Z 940.063,A -85,B 0,C 180,E1 968.524,E2 968.524} C_VEL
LIN {X 0,Y 602.262,Z 966.927,A -85,B 0,C 180,E1 972.064,E2 972.064} C_VEL
LIN {X 0,Y 602.163,Z 988.719,A -85,B 0,C 180,E1 975.809,E2 975.809} C_VEL
LIN {X 0,Y 602.064,Z 1004.736,A -85,B 0,C 180,E1 979.577,E2 979.577} C_VEL
LIN {X 0,Y 602.051,Z 1014.332,A -85,B 0,C 180,E1 982.777,E2 982.777} C_VEL
LIN {X 0,Y 602.18,Z 1019.905,A -85,B 0,C 180,E1 985.674,E2 985.674} C_VEL
LIN {X 0,Y 602.207,Z 1022.657,A -85,B 0,C 180,E1 988.56,E2 988.56} C_VEL
LIN {X 0,Y 602.154,Z 1021.627,A -85,B 0,C 180,E1 992.883,E2 992.883} C_VEL
LIN {X 0,Y 602.18,Z 1014.331,A -85,B 0,C 180,E1 997.222,E2 997.222} C_VEL
LIN {X 0,Y 602.131,Z 1001.486,A -85,B 0,C 180,E1 1001.305,E2 1001.305} C_VEL
LIN {X 0,Y 602.203,Z 982.822,A -85,B 0,C 180,E1 1005.308,E2 1005.308} C_VEL
LIN {X 0,Y 602.333,Z 959.01,A -85,B 0,C 180,E1 1009.074,E2 1009.074} C_VEL
LIN {X 0,Y 602.632,Z 931.01,A -85,B 0,C 180,E1 1012.489,E2 1012.489} C_VEL
LIN {X 0,Y 602.982,Z 898.187,A -85,B 0,C 180,E1 1015.627,E2 1015.627} C_VEL
LIN {X 0,Y 603.416,Z 861.13,A -85,B 0,C 180,E1 1018.373,E2 1018.373} C_VEL
LIN {X 0,Y 603.797,Z 822.167,A -85,B 0,C 180,E1 1020.548,E2 1020.548} C_VEL
LIN {X 0,Y 604.148,Z 783.88,A -85,B 0,C 180,E1 1022.086,E2 1022.086} C_VEL
LIN {X 0,Y 604.346,Z 747.424,A -85,B 0,C 180,E1 1023.054,E2 1023.054} C_VEL
LIN {X 0,Y 603.4,Z 695.855,A -85,B 0,C 180,E1 1023.901,E2 1023.901} C_VEL
LIN {X 0,Y 601.973,Z 691.44,A -85,B 0,C 180,E1 1024.105,E2 1024.105} C_VEL
LIN {X 0,Y 601.759,Z 691.44,A -85,B 0,C 180,E1 1028.979,E2 1028.979} C_VEL
LIN {X 0,Y 601.716,Z 691.44,A -85,B 0,C 180,E1 1035.209,E2 1035.209} C_VEL
LIN {X 0,Y 601.735,Z 691.44,A -85,B 0,C 180,E1 1041.263,E2 1041.263} C_VEL
LIN {X 0,Y 601.526,Z 691.44,A -85,B 0,C 180,E1 1046.376,E2 1046.376} C_VEL
LIN {X 0,Y 601.633,Z 691.44,A -85,B 0,C 180,E1 1051.435,E2 1051.435} C_VEL
LIN {X 0,Y 601.704,Z 691.44,A -85,B 0,C 180,E1 1056.258,E2 1056.258} C_VEL
LIN {X 0,Y 601.9,Z 691.44,A -85,B 0,C 180,E1 1060.911,E2 1060.911} C_VEL
LIN {X 0,Y 601.485,Z 691.44,A -85,B 0,C 180,E1 1065.419,E2 1065.419} C_VEL
LIN {X 0,Y 601.923,Z 691.44,A -85,B 0,C 180,E1 1069.856,E2 1069.856} C_VEL
LIN {X 0,Y 602.156,Z 691.44,A -85,B 0,C 180,E1 1074.225,E2 1074.225} C_VEL
LIN {X 0,Y 601.868,Z 691.44,A -85,B 0,C 180,E1 1079.997,E2 1079.997} C_VEL
LIN {X 0,Y 601.905,Z 691.44,A -85,B 0,C 180,E1 1084.324,E2 1084.324} C_VEL
LIN {X 0,Y 601.973,Z 691.44,A -85,B 0,C 180,E1 1088.675,E2 1088.675} C_VEL
LIN {X 0,Y 602.075,Z 691.44,A -85,B 0,C 180,E1 1093.076,E2 1093.076} C_VEL
LIN {X 0,Y 601.835,Z 691.44,A -85,B 0,C 180,E1 1099.083,E2 1099.083} C_VEL
LIN {X 0,Y 601.754,Z 691.44,A -85,B 0,C 180,E1 1103.732,E2 1103.732} C_VEL
LIN {X 0,Y 601.786,Z 691.44,A -85,B 0,C 180,E1 1108.549,E2 1108.549} C_VEL
LIN {X 0,Y 601.924,Z 691.44,A -85,B 0,C 180,E1 1113.892,E2 1113.892} C_VEL
LIN {X 0,Y 601.719,Z 691.44,A -85,B 0,C 180,E1 1118.97,E2 1118.97} C_VEL
LIN {X 0,Y 601.596,Z 691.44,A -85,B 0,C 180,E1 1123.124,E2 1123.124} C_VEL
LIN {X 0,Y 601.746,Z 691.44,A -85,B 0,C 180,E1 1129.141,E2 1129.141} C_VEL
LIN {X 0,Y 601.88,Z 691.44,A -85,B 0,C 180,E1 1134.648,E2 1134.648} C_VEL
LIN {X 0,Y 601.966,Z 691.44,A -85,B 0,C 180,E1 1136.295,E2 1136.295} C_VEL
LIN {X 0,Y 604.218,Z 702.818,A -85,B 0,C 180,E1 1136.632,E2 1136.632} C_VEL
LIN {X 0,Y 604.217,Z 744.355,A -85,B 0,C 180,E1 1137.564,E2 1137.564} C_VEL
LIN {X 0,Y 603.884,Z 786.185,A -85,B 0,C 180,E1 1139.125,E2 1139.125} C_VEL
LIN {X 0,Y 603.478,Z 825.967,A -85,B 0,C 180,E1 1141.256,E2 1141.256} C_VEL
LIN {X 0,Y 603.02,Z 863.469,A -85,B 0,C 180,E1 1143.935,E2 1143.935} C_VEL
LIN {X 0,Y 602.686,Z 898.187,A -85,B 0,C 180,E1 1147.157,E2 1147.157} C_VEL
LIN {X 0,Y 602.384,Z 928.178,A -85,B 0,C 180,E1 1150.765,E2 1150.765} C_VEL
LIN {X 0,Y 602.183,Z 952.073,A -85,B 0,C 180,E1 1154.505,E2 1154.505} C_VEL
LIN {X 0,Y 602.111,Z 970.497,A -85,B 0,C 180,E1 1158.394,E2 1158.394} C_VEL
LIN {X 0,Y 602.053,Z 982.52,A -85,B 0,C 180,E1 1162.049,E2 1162.049} C_VEL
LIN {X 0,Y 602.032,Z 989.969,A -85,B 0,C 180,E1 1165.673,E2 1165.673} C_VEL
LIN {X 0,Y 602.018,Z 992.677,A -85,B 0,C 180,E1 1168.559,E2 1168.559} C_VEL
LIN {X 0,Y 602.142,Z 992.629,A -85,B 0,C 180,E1 1171.441,E2 1171.441} C_VEL
LIN {X 0,Y 602.196,Z 987.384,A -85,B 0,C 180,E1 1175.772,E2 1175.772} C_VEL
LIN {X 0,Y 602.203,Z 976.838,A -85,B 0,C 180,E1 1179.771,E2 1179.771} C_VEL
LIN {X 0,Y 602.207,Z 960.266,A -85,B 0,C 180,E1 1183.818,E2 1183.818} C_VEL
LIN {X 0,Y 602.295,Z 939.071,A -85,B 0,C 180,E1 1187.557,E2 1187.557} C_VEL
LIN {X 0,Y 602.527,Z 912.688,A -85,B 0,C 180,E1 1191.116,E2 1191.116} C_VEL
LIN {X 0,Y 602.861,Z 881.663,A -85,B 0,C 180,E1 1194.382,E2 1194.382} C_VEL
LIN {X 0,Y 603.218,Z 848.3,A -85,B 0,C 180,E1 1197.142,E2 1197.142} C_VEL
LIN {X 0,Y 603.587,Z 810.845,A -85,B 0,C 180,E1 1199.543,E2 1199.543} C_VEL
LIN {X 0,Y 603.915,Z 771.517,A -85,B 0,C 180,E1 1201.411,E2 1201.411} C_VEL
LIN {X 0,Y 604.317,Z 729.501,A -85,B 0,C 180,E1 1202.745,E2 1202.745} C_VEL
LIN {X 0,Y 603.511,Z 695.912,A -85,B 0,C 180,E1 1203.428,E2 1203.428} C_VEL
LIN {X 0,Y 602.031,Z 691.44,A -85,B 0,C 180,E1 1203.593,E2 1203.593} C_VEL
LIN {X 0,Y 601.749,Z 691.44,A -85,B 0,C 180,E1 1208.979,E2 1208.979} C_VEL
LIN {X 0,Y 601.715,Z 691.44,A -85,B 0,C 180,E1 1215.219,E2 1215.219} C_VEL
LIN {X 0,Y 601.669,Z 691.44,A -85,B 0,C 180,E1 1221.026,E2 1221.026} C_VEL
LIN {X 0,Y 601.539,Z 691.44,A -85,B 0,C 180,E1 1226.162,E2 1226.162} C_VEL
LIN {X 0,Y 601.64,Z 691.44,A -85,B 0,C 180,E1 1231.443,E2 1231.443} C_VEL
LIN {X 0,Y 601.749,Z 691.44,A -85,B 0,C 180,E1 1236.268,E2 1236.268} C_VEL
LIN {X 0,Y 601.927,Z 691.44,A -85,B 0,C 180,E1 1240.92,E2 1240.92} C_VEL
LIN {X 0,Y 602.133,Z 691.44,A -85,B 0,C 180,E1 1246.926,E2 1246.926} C_VEL
LIN {X 0,Y 601.85,Z 691.44,A -85,B 0,C 180,E1 1252.778,E2 1252.778} C_VEL
LIN {X 0,Y 601.857,Z 691.44,A -85,B 0,C 180,E1 1257.631,E2 1257.631} C_VEL
LIN {X 0,Y 597.806,Z 691.44,A -85,B 0,C 180,E1 1259.255,E2 1259.255} C_VEL
LIN {X 0,Y 594.089,Z 691.44,A -85,B 0,C 180,E1 1260.901,E2 1260.901} C_VEL
LIN {X 0,Y 594.062,Z 691.44,A -85,B 0,C 180,E1 1266.286,E2 1266.286} C_VEL
LIN {X 0,Y 593.884,Z 691.44,A -85,B 0,C 180,E1 1271.77,E2 1271.77} C_VEL
LIN {X 0,Y 593.884,Z 691.44,A -85,B 0,C 180,E1 1276.288,E2 1276.288} C_VEL
LIN {X 0,Y 593.941,Z 691.44,A -85,B 0,C 180,E1 1280.91,E2 1280.91} C_VEL
LIN {X 0,Y 593.953,Z 691.44,A -85,B 0,C 180,E1 1285.681,E2 1285.681} C_VEL
LIN {X 0,Y 593.802,Z 691.44,A -85,B 0,C 180,E1 1290.661,E2 1290.661} C_VEL
LIN {X 0,Y 593.852,Z 691.44,A -85,B 0,C 180,E1 1295.901,E2 1295.901} C_VEL
LIN {X 0,Y 593.775,Z 691.44,A -85,B 0,C 180,E1 1301.525,E2 1301.525} C_VEL
LIN {X 0,Y 593.685,Z 691.44,A -85,B 0,C 180,E1 1306.482,E2 1306.482} C_VEL
LIN {X 0,Y 593.688,Z 691.44,A -85,B 0,C 180,E1 1312.261,E2 1312.261} C_VEL
LIN {X 0,Y 593.891,Z 691.751,A -85,B 0,C 180,E1 1315.421,E2 1315.421} C_VEL
LIN {X 0,Y 597.435,Z 700.305,A -85,B 0,C 180,E1 1315.777,E2 1315.777} C_VEL
LIN {X 0,Y 597.545,Z 758.798,A -85,B 0,C 180,E1 1316.773,E2 1316.773} C_VEL
LIN {X 0,Y 597.148,Z 799.226,A -85,B 0,C 180,E1 1318.057,E2 1318.057} C_VEL
LIN {X 0,Y 596.561,Z 838.847,A -85,B 0,C 180,E1 1319.917,E2 1319.917} C_VEL
LIN {X 0,Y 596.013,Z 875.092,A -85,B 0,C 180,E1 1322.217,E2 1322.217} C_VEL
LIN {X 0,Y 595.378,Z 909.882,A -85,B 0,C 180,E1 1325.074,E2 1325.074} C_VEL
LIN {X 0,Y 594.88,Z 940.065,A -85,B 0,C 180,E1 1328.234,E2 1328.234} C_VEL
LIN {X 0,Y 594.515,Z 966.929,A -85,B 0,C 180,E1 1331.822,E2 1331.822} C_VEL
LIN {X 0,Y 594.32,Z 987.959,A -85,B 0,C 180,E1 1335.469,E2 1335.469} C_VEL
LIN {X 0,Y 594.195,Z 1003.951,A -85,B 0,C 180,E1 1339.222,E2 1339.222} C_VEL
LIN {X 0,Y 594.161,Z 1014.332,A -85,B 0,C 180,E1 1342.68,E2 1342.68} C_VEL
LIN {X 0,Y 594.283,Z 1019.905,A -85,B 0,C 180,E1 1345.617,E2 1345.617} C_VEL
LIN {X 0,Y 594.3,Z 1022.657,A -85,B 0,C 180,E1 1348.54,E2 1348.54} C_VEL
LIN {X 0,Y 594.247,Z 1021.627,A -85,B 0,C 180,E1 1352.921,E2 1352.921} C_VEL
LIN {X 0,Y 594.294,Z 1014.331,A -85,B 0,C 180,E1 1357.319,E2 1357.319} C_VEL
LIN {X 0,Y 594.272,Z 1002.017,A -85,B 0,C 180,E1 1361.311,E2 1361.311} C_VEL
LIN {X 0,Y 594.399,Z 984.795,A -85,B 0,C 180,E1 1365.135,E2 1365.135} C_VEL
LIN {X 0,Y 594.614,Z 963.036,A -85,B 0,C 180,E1 1368.752,E2 1368.752} C_VEL
LIN {X 0,Y 595,Z 935.613,A -85,B 0,C 180,E1 1372.278,E2 1372.278} C_VEL
LIN {X 0,Y 595.49,Z 903.732,A -85,B 0,C 180,E1 1375.484,E2 1375.484} C_VEL
LIN {X 0,Y 596.142,Z 868.26,A -85,B 0,C 180,E1 1378.265,E2 1378.265} C_VEL
LIN {X 0,Y 596.731,Z 829.796,A -85,B 0,C 180,E1 1380.569,E2 1380.569} C_VEL
LIN {X 0,Y 597.364,Z 789.667,A -85,B 0,C 180,E1 1382.298,E2 1382.298} C_VEL
LIN {X 0,Y 597.663,Z 750.995,A -85,B 0,C 180,E1 1383.393,E2 1383.393} C_VEL
LIN {X 0,Y 597.167,Z 699.391,A -85,B 0,C 180,E1 1384.253,E2 1384.253} C_VEL
LIN {X 0,Y 593.886,Z 691.44,A -85,B 0,C 180,E1 1384.632,E2 1384.632} C_VEL
LIN {X 0,Y 593.68,Z 691.44,A -85,B 0,C 180,E1 1390.088,E2 1390.088} C_VEL
LIN {X 0,Y 593.785,Z 691.44,A -85,B 0,C 180,E1 1395.559,E2 1395.559} C_VEL
LIN {X 0,Y 593.728,Z 691.44,A -85,B 0,C 180,E1 1400.394,E2 1400.394} C_VEL
LIN {X 0,Y 593.662,Z 691.44,A -85,B 0,C 180,E1 1405.87,E2 1405.87} C_VEL
LIN {X 0,Y 593.723,Z 691.44,A -85,B 0,C 180,E1 1411.019,E2 1411.019} C_VEL
LIN {X 0,Y 593.877,Z 691.44,A -85,B 0,C 180,E1 1415.926,E2 1415.926} C_VEL
LIN {X 0,Y 593.988,Z 691.44,A -85,B 0,C 180,E1 1420.647,E2 1420.647} C_VEL
LIN {X 0,Y 593.63,Z 691.44,A -85,B 0,C 180,E1 1425.222,E2 1425.222} C_VEL
LIN {X 0,Y 593.985,Z 691.44,A -85,B 0,C 180,E1 1429.719,E2 1429.719} C_VEL
LIN {X 0,Y 594.218,Z 691.44,A -85,B 0,C 180,E1 1434.147,E2 1434.147} C_VEL
LIN {X 0,Y 593.968,Z 691.44,A -85,B 0,C 180,E1 1439.996,E2 1439.996} C_VEL
LIN {X 0,Y 593.989,Z 691.44,A -85,B 0,C 180,E1 1444.382,E2 1444.382} C_VEL
LIN {X 0,Y 594.056,Z 691.44,A -85,B 0,C 180,E1 1448.792,E2 1448.792} C_VEL
LIN {X 0,Y 593.872,Z 691.44,A -85,B 0,C 180,E1 1454.345,E2 1454.345} C_VEL
LIN {X 0,Y 593.892,Z 691.44,A -85,B 0,C 180,E1 1459.388,E2 1459.388} C_VEL
LIN {X 0,Y 593.827,Z 691.44,A -85,B 0,C 180,E1 1464.069,E2 1464.069} C_VEL
LIN {X 0,Y 593.79,Z 691.44,A -85,B 0,C 180,E1 1468.97,E2 1468.97} C_VEL
LIN {X 0,Y 594,Z 691.44,A -85,B 0,C 180,E1 1474.1,E2 1474.1} C_VEL
LIN {X 0,Y 593.758,Z 691.44,A -85,B 0,C 180,E1 1480.093,E2 1480.093} C_VEL
LIN {X 0,Y 593.55,Z 691.44,A -85,B 0,C 180,E1 1485.569,E2 1485.569} C_VEL
LIN {X 0,Y 593.767,Z 691.44,A -85,B 0,C 180,E1 1490.395,E2 1490.395} C_VEL
LIN {X 0,Y 594.056,Z 691.44,A -85,B 0,C 180,E1 1495.779,E2 1495.779} C_VEL
LIN {X 0,Y 597.429,Z 701.993,A -85,B 0,C 180,E1 1496.189,E2 1496.189} C_VEL
LIN {X 0,Y 597.438,Z 744.836,A -85,B 0,C 180,E1 1497.167,E2 1497.167} C_VEL
LIN {X 0,Y 596.953,Z 787.104,A -85,B 0,C 180,E1 1498.768,E2 1498.768} C_VEL
LIN {X 0,Y 596.338,Z 826.194,A -85,B 0,C 180,E1 1500.893,E2 1500.893} C_VEL
LIN {X 0,Y 595.671,Z 863.453,A -85,B 0,C 180,E1 1503.588,E2 1503.588} C_VEL
LIN {X 0,Y 595.101,Z 897.447,A -85,B 0,C 180,E1 1506.773,E2 1506.773} C_VEL
LIN {X 0,Y 594.645,Z 927.263,A -85,B 0,C 180,E1 1510.373,E2 1510.373} C_VEL
LIN {X 0,Y 594.364,Z 951.034,A -85,B 0,C 180,E1 1514.106,E2 1514.106} C_VEL
LIN {X 0,Y 594.202,Z 968.948,A -85,B 0,C 180,E1 1517.865,E2 1517.865} C_VEL
LIN {X 0,Y 594.18,Z 980.575,A -85,B 0,C 180,E1 1521.205,E2 1521.205} C_VEL
LIN {X 0,Y 594.154,Z 988.775,A -85,B 0,C 180,E1 1524.883,E2 1524.883} C_VEL
LIN {X 0,Y 594.119,Z 992.677,A -85,B 0,C 180,E1 1528.539,E2 1528.539} C_VEL
LIN {X 0,Y 594.237,Z 992.629,A -85,B 0,C 180,E1 1531.46,E2 1531.46} C_VEL
LIN {X 0,Y 594.284,Z 987.385,A -85,B 0,C 180,E1 1535.849,E2 1535.849} C_VEL
LIN {X 0,Y 594.313,Z 976.841,A -85,B 0,C 180,E1 1539.902,E2 1539.902} C_VEL
LIN {X 0,Y 594.352,Z 960.766,A -85,B 0,C 180,E1 1543.899,E2 1543.899} C_VEL
LIN {X 0,Y 594.504,Z 940.079,A -85,B 0,C 180,E1 1547.637,E2 1547.637} C_VEL
LIN {X 0,Y 594.868,Z 915.161,A -85,B 0,C 180,E1 1551.102,E2 1551.102} C_VEL
LIN {X 0,Y 595.354,Z 885.091,A -85,B 0,C 180,E1 1554.383,E2 1554.383} C_VEL
LIN {X 0,Y 595.88,Z 850.941,A -85,B 0,C 180,E1 1557.309,E2 1557.309} C_VEL
LIN {X 0,Y 596.509,Z 812.699,A -85,B 0,C 180,E1 1559.826,E2 1559.826} C_VEL
LIN {X 0,Y 597.089,Z 771.539,A -85,B 0,C 180,E1 1561.812,E2 1561.812} C_VEL
LIN {X 0,Y 597.633,Z 729.912,A -85,B 0,C 180,E1 1563.147,E2 1563.147} C_VEL
LIN {X 0,Y 597.284,Z 699.591,A -85,B 0,C 180,E1 1563.77,E2 1563.77} C_VEL
LIN {X 0,Y 593.973,Z 691.44,A -85,B 0,C 180,E1 1564.111,E2 1564.111} C_VEL
LIN {X 0,Y 593.664,Z 691.44,A -85,B 0,C 180,E1 1570.097,E2 1570.097} C_VEL
LIN {X 0,Y 593.784,Z 691.44,A -85,B 0,C 180,E1 1575.558,E2 1575.558} C_VEL
LIN {X 0,Y 593.71,Z 691.44,A -85,B 0,C 180,E1 1580.402,E2 1580.402} C_VEL
LIN {X 0,Y 593.654,Z 691.44,A -85,B 0,C 180,E1 1585.878,E2 1585.878} C_VEL
LIN {X 0,Y 593.728,Z 691.44,A -85,B 0,C 180,E1 1591.027,E2 1591.027} C_VEL
LIN {X 0,Y 593.908,Z 691.44,A -85,B 0,C 180,E1 1595.935,E2 1595.935} C_VEL
LIN {X 0,Y 594.012,Z 691.44,A -85,B 0,C 180,E1 1600.655,E2 1600.655} C_VEL
LIN {X 0,Y 594.191,Z 691.44,A -85,B 0,C 180,E1 1606.748,E2 1606.748} C_VEL
LIN {X 0,Y 593.967,Z 691.44,A -85,B 0,C 180,E1 1612.682,E2 1612.682} C_VEL
LIN {X 0,Y 593.949,Z 691.44,A -85,B 0,C 180,E1 1617.616,E2 1617.616} C_VEL
LIN {X 0,Y 594.089,Z 691.44,A -85,B 0,C 180,E1 1620.901,E2 1620.901} C_VEL
LIN {X 0,Y 591.579,Z 691.44,A -85,B 0,C 180,E1 1622.145,E2 1622.145} C_VEL
LIN {X 0,Y 586.059,Z 691.44,A -85,B 0,C 180,E1 1624.005,E2 1624.005} C_VEL
LIN {X 0,Y 585.981,Z 691.44,A -85,B 0,C 180,E1 1624.221,E2 1624.221} C_VEL
LIN {X 0,Y 585.896,Z 691.44,A -85,B 0,C 180,E1 1628.922,E2 1628.922} C_VEL
LIN {X 0,Y 585.926,Z 691.44,A -85,B 0,C 180,E1 1633.45,E2 1633.45} C_VEL
LIN {X 0,Y 585.829,Z 691.44,A -85,B 0,C 180,E1 1638.069,E2 1638.069} C_VEL
LIN {X 0,Y 585.849,Z 691.44,A -85,B 0,C 180,E1 1642.81,E2 1642.81} C_VEL
LIN {X 0,Y 585.774,Z 691.44,A -85,B 0,C 180,E1 1647.727,E2 1647.727} C_VEL
LIN {X 0,Y 585.706,Z 691.44,A -85,B 0,C 180,E1 1652.878,E2 1652.878} C_VEL
LIN {X 0,Y 585.84,Z 691.44,A -85,B 0,C 180,E1 1658.334,E2 1658.334} C_VEL
LIN {X 0,Y 585.893,Z 691.44,A -85,B 0,C 180,E1 1664.243,E2 1664.243} C_VEL
LIN {X 0,Y 585.781,Z 691.44,A -85,B 0,C 180,E1 1669.746,E2 1669.746} C_VEL
LIN {X 0,Y 585.852,Z 691.762,A -85,B 0,C 180,E1 1674.878,E2 1674.878} C_VEL
LIN {X 0,Y 591.002,Z 702.806,A -85,B 0,C 180,E1 1675.388,E2 1675.388} C_VEL
LIN {X 0,Y 590.898,Z 759.038,A -85,B 0,C 180,E1 1676.355,E2 1676.355} C_VEL
LIN {X 0,Y 590.34,Z 801.013,A -85,B 0,C 180,E1 1677.714,E2 1677.714} C_VEL
LIN {X 0,Y 589.52,Z 840.608,A -85,B 0,C 180,E1 1679.619,E2 1679.619} C_VEL
LIN {X 0,Y 588.708,Z 877.738,A -85,B 0,C 180,E1 1682.042,E2 1682.042} C_VEL
LIN {X 0,Y 587.894,Z 911.141,A -85,B 0,C 180,E1 1684.858,E2 1684.858} C_VEL
LIN {X 0,Y 587.228,Z 941.776,A -85,B 0,C 180,E1 1688.147,E2 1688.147} C_VEL
LIN {X 0,Y 586.753,Z 966.931,A -85,B 0,C 180,E1 1691.573,E2 1691.573} C_VEL
LIN {X 0,Y 586.484,Z 988.621,A -85,B 0,C 180,E1 1695.401,E2 1695.401} C_VEL
LIN {X 0,Y 586.339,Z 1004.504,A -85,B 0,C 180,E1 1699.229,E2 1699.229} C_VEL
LIN {X 0,Y 586.271,Z 1014.332,A -85,B 0,C 180,E1 1702.581,E2 1702.581} C_VEL
LIN {X 0,Y 586.386,Z 1019.905,A -85,B 0,C 180,E1 1705.558,E2 1705.558} C_VEL
LIN {X 0,Y 586.395,Z 1022.657,A -85,B 0,C 180,E1 1708.521,E2 1708.521} C_VEL
LIN {X 0,Y 586.343,Z 1021.627,A -85,B 0,C 180,E1 1712.961,E2 1712.961} C_VEL
LIN {X 0,Y 586.381,Z 1014.33,A -85,B 0,C 180,E1 1717.418,E2 1717.418} C_VEL
LIN {X 0,Y 586.38,Z 1001.999,A -85,B 0,C 180,E1 1721.47,E2 1721.47} C_VEL
LIN {X 0,Y 586.546,Z 984.797,A -85,B 0,C 180,E1 1725.343,E2 1725.343} C_VEL
LIN {X 0,Y 586.861,Z 963.038,A -85,B 0,C 180,E1 1729.01,E2 1729.01} C_VEL
LIN {X 0,Y 587.417,Z 935.279,A -85,B 0,C 180,E1 1732.619,E2 1732.619} C_VEL
LIN {X 0,Y 588.108,Z 903.72,A -85,B 0,C 180,E1 1735.828,E2 1735.828} C_VEL
LIN {X 0,Y 588.913,Z 868.672,A -85,B 0,C 180,E1 1738.616,E2 1738.616} C_VEL
LIN {X 0,Y 589.786,Z 829.674,A -85,B 0,C 180,E1 1740.974,E2 1740.974} C_VEL
LIN {X 0,Y 590.607,Z 789.197,A -85,B 0,C 180,E1 1742.731,E2 1742.731} C_VEL
LIN {X 0,Y 591.084,Z 750.637,A -85,B 0,C 180,E1 1743.823,E2 1743.823} C_VEL
LIN {X 0,Y 590.428,Z 701.496,A -85,B 0,C 180,E1 1744.669,E2 1744.669} C_VEL
LIN {X 0,Y 585.853,Z 691.44,A -85,B 0,C 180,E1 1745.175,E2 1745.175} C_VEL
LIN {X 0,Y 585.785,Z 691.44,A -85,B 0,C 180,E1 1750.254,E2 1750.254} C_VEL
LIN {X 0,Y 585.915,Z 691.44,A -85,B 0,C 180,E1 1756.349,E2 1756.349} C_VEL
LIN {X 0,Y 585.842,Z 691.44,A -85,B 0,C 180,E1 1761.666,E2 1761.666} C_VEL
LIN {X 0,Y 585.718,Z 691.44,A -85,B 0,C 180,E1 1767.123,E2 1767.123} C_VEL
LIN {X 0,Y 585.763,Z 691.44,A -85,B 0,C 180,E1 1772.273,E2 1772.273} C_VEL
LIN {X 0,Y 585.834,Z 691.44,A -85,B 0,C 180,E1 1777.19,E2 1777.19} C_VEL
LIN {X 0,Y 586.058,Z 691.44,A -85,B 0,C 180,E1 1781.938,E2 1781.938} C_VEL
LIN {X 0,Y 585.763,Z 691.44,A -85,B 0,C 180,E1 1788.064,E2 1788.064} C_VEL
LIN {X 0,Y 586.293,Z 691.44,A -85,B 0,C 180,E1 1794.068,E2 1794.068} C_VEL
LIN {X 0,Y 586.078,Z 691.44,A -85,B 0,C 180,E1 1799.996,E2 1799.996} C_VEL
LIN {X 0,Y 586.084,Z 691.44,A -85,B 0,C 180,E1 1804.441,E2 1804.441} C_VEL
LIN {X 0,Y 586.119,Z 691.44,A -85,B 0,C 180,E1 1808.912,E2 1808.912} C_VEL
LIN {X 0,Y 586.166,Z 691.44,A -85,B 0,C 180,E1 1813.437,E2 1813.437} C_VEL
LIN {X 0,Y 585.982,Z 691.44,A -85,B 0,C 180,E1 1819.621,E2 1819.621} C_VEL
LIN {X 0,Y 585.863,Z 691.44,A -85,B 0,C 180,E1 1824.417,E2 1824.417} C_VEL
LIN {X 0,Y 585.827,Z 691.44,A -85,B 0,C 180,E1 1829.402,E2 1829.402} C_VEL
LIN {X 0,Y 586.041,Z 691.44,A -85,B 0,C 180,E1 1834.628,E2 1834.628} C_VEL
LIN {X 0,Y 585.869,Z 691.44,A -85,B 0,C 180,E1 1840.236,E2 1840.236} C_VEL
LIN {X 0,Y 585.742,Z 691.44,A -85,B 0,C 180,E1 1846.353,E2 1846.353} C_VEL
LIN {X 0,Y 585.882,Z 691.44,A -85,B 0,C 180,E1 1851.667,E2 1851.667} C_VEL
LIN {X 0,Y 586.102,Z 691.44,A -85,B 0,C 180,E1 1855.277,E2 1855.277} C_VEL
LIN {X 0,Y 590.937,Z 704.169,A -85,B 0,C 180,E1 1855.805,E2 1855.805} C_VEL
LIN {X 0,Y 590.714,Z 746.406,A -85,B 0,C 180,E1 1856.798,E2 1856.798} C_VEL
LIN {X 0,Y 590.063,Z 787.385,A -85,B 0,C 180,E1 1858.375,E2 1858.375} C_VEL
LIN {X 0,Y 589.208,Z 827.791,A -85,B 0,C 180,E1 1860.607,E2 1860.607} C_VEL
LIN {X 0,Y 588.27,Z 865.708,A -85,B 0,C 180,E1 1863.417,E2 1863.417} C_VEL
LIN {X 0,Y 587.514,Z 899.604,A -85,B 0,C 180,E1 1866.694,E2 1866.694} C_VEL
LIN {X 0,Y 586.913,Z 928.291,A -85,B 0,C 180,E1 1870.254,E2 1870.254} C_VEL
LIN {X 0,Y 586.533,Z 952.069,A -85,B 0,C 180,E1 1874.081,E2 1874.081} C_VEL
LIN {X 0,Y 586.355,Z 970.491,A -85,B 0,C 180,E1 1878.078,E2 1878.078} C_VEL
LIN {X 0,Y 586.286,Z 982.518,A -85,B 0,C 180,E1 1881.834,E2 1881.834} C_VEL
LIN {X 0,Y 586.23,Z 989.968,A -85,B 0,C 180,E1 1885.556,E2 1885.556} C_VEL
LIN {X 0,Y 586.226,Z 992.677,A -85,B 0,C 180,E1 1888.52,E2 1888.52} C_VEL
LIN {X 0,Y 586.332,Z 992.63,A -85,B 0,C 180,E1 1891.479,E2 1891.479} C_VEL
LIN {X 0,Y 586.371,Z 987.387,A -85,B 0,C 180,E1 1895.928,E2 1895.928} C_VEL
LIN {X 0,Y 586.41,Z 976.843,A -85,B 0,C 180,E1 1900.037,E2 1900.037} C_VEL
LIN {X 0,Y 586.486,Z 961.053,A -85,B 0,C 180,E1 1904.028,E2 1904.028} C_VEL
LIN {X 0,Y 586.746,Z 940.372,A -85,B 0,C 180,E1 1907.833,E2 1907.833} C_VEL
LIN {X 0,Y 587.223,Z 914.141,A -85,B 0,C 180,E1 1911.517,E2 1911.517} C_VEL
LIN {X 0,Y 587.87,Z 883.613,A -85,B 0,C 180,E1 1914.858,E2 1914.858} C_VEL
LIN {X 0,Y 588.642,Z 849.626,A -85,B 0,C 180,E1 1917.774,E2 1917.774} C_VEL
LIN {X 0,Y 589.515,Z 812.6,A -85,B 0,C 180,E1 1920.223,E2 1920.223} C_VEL
LIN {X 0,Y 590.307,Z 772.236,A -85,B 0,C 180,E1 1922.195,E2 1922.195} C_VEL
LIN {X 0,Y 590.959,Z 730.987,A -85,B 0,C 180,E1 1923.542,E2 1923.542} C_VEL
LIN {X 0,Y 590.481,Z 701.592,A -85,B 0,C 180,E1 1924.179,E2 1924.179} C_VEL
LIN {X 0,Y 585.941,Z 691.44,A -85,B 0,C 180,E1 1924.644,E2 1924.644} C_VEL
LIN {X 0,Y 585.769,Z 691.44,A -85,B 0,C 180,E1 1930.255,E2 1930.255} C_VEL
LIN {X 0,Y 585.907,Z 691.44,A -85,B 0,C 180,E1 1936.349,E2 1936.349} C_VEL
LIN {X 0,Y 585.803,Z 691.44,A -85,B 0,C 180,E1 1941.672,E2 1941.672} C_VEL
LIN {X 0,Y 585.709,Z 691.44,A -85,B 0,C 180,E1 1947.131,E2 1947.131} C_VEL
LIN {X 0,Y 585.781,Z 691.44,A -85,B 0,C 180,E1 1952.282,E2 1952.282} C_VEL
LIN {X 0,Y 585.862,Z 691.44,A -85,B 0,C 180,E1 1957.199,E2 1957.199} C_VEL
LIN {X 0,Y 586.025,Z 691.44,A -85,B 0,C 180,E1 1961.945,E2 1961.945} C_VEL
LIN {X 0,Y 586.264,Z 691.44,A -85,B 0,C 180,E1 1966.565,E2 1966.565} C_VEL
LIN {X 0,Y 586.064,Z 691.44,A -85,B 0,C 180,E1 1972.583,E2 1972.583} C_VEL
LIN {X 0,Y 586.193,Z 691.44,A -85,B 0,C 180,E1 1977.043,E2 1977.043} C_VEL
LIN {X 0,Y 586.324,Z 691.44,A -85,B 0,C 180,E1 1981.483,E2 1981.483} C_VEL
LIN {X 0,Y 585.981,Z 691.44,A -85,B 0,C 180,E1 1984.221,E2 1984.221} C_VEL
LIN {X 0,Y 583.546,Z 691.44,A -85,B 0,C 180,E1 1985.484,E2 1985.484} C_VEL
LIN {X 0,Y 578.03,Z 691.44,A -85,B 0,C 180,E1 1987.593,E2 1987.593} C_VEL
LIN {X 0,Y 578.057,Z 691.44,A -85,B 0,C 180,E1 1992.097,E2 1992.097} C_VEL
LIN {X 0,Y 578.018,Z 691.44,A -85,B 0,C 180,E1 1996.748,E2 1996.748} C_VEL
LIN {X 0,Y 578.035,Z 691.44,A -85,B 0,C 180,E1 2001.514,E2 2001.514} C_VEL
LIN {X 0,Y 577.924,Z 691.44,A -85,B 0,C 180,E1 2007.032,E2 2007.032} C_VEL
LIN {X 0,Y 577.819,Z 691.44,A -85,B 0,C 180,E1 2013.018,E2 2013.018} C_VEL
LIN {X 0,Y 577.926,Z 691.44,A -85,B 0,C 180,E1 2018.191,E2 2018.191} C_VEL
LIN {X 0,Y 577.954,Z 691.44,A -85,B 0,C 180,E1 2022.93,E2 2022.93} C_VEL
LIN {X 0,Y 577.82,Z 691.44,A -85,B 0,C 180,E1 2029.074,E2 2029.074} C_VEL
LIN {X 0,Y 577.869,Z 691.44,A -85,B 0,C 180,E1 2034.31,E2 2034.31} C_VEL
LIN {X 0,Y 584.137,Z 705.072,A -85,B 0,C 180,E1 2034.955,E2 2034.955} C_VEL
LIN {X 0,Y 584.269,Z 760.497,A -85,B 0,C 180,E1 2035.963,E2 2035.963} C_VEL
LIN {X 0,Y 583.544,Z 802.505,A -85,B 0,C 180,E1 2037.351,E2 2037.351} C_VEL
LIN {X 0,Y 582.492,Z 843.419,A -85,B 0,C 180,E1 2039.374,E2 2039.374} C_VEL
LIN {X 0,Y 581.36,Z 881.704,A -85,B 0,C 180,E1 2041.962,E2 2041.962} C_VEL
LIN {X 0,Y 580.286,Z 917.93,A -85,B 0,C 180,E1 2045.175,E2 2045.175} C_VEL
LIN {X 0,Y 579.498,Z 948.915,A -85,B 0,C 180,E1 2048.745,E2 2048.745} C_VEL
LIN {X 0,Y 578.974,Z 975.057,A -85,B 0,C 180,E1 2052.653,E2 2052.653} C_VEL
LIN {X 0,Y 578.658,Z 995.669,A -85,B 0,C 180,E1 2056.765,E2 2056.765} C_VEL
LIN {X 0,Y 578.555,Z 1010.441,A -85,B 0,C 180,E1 2060.966,E2 2060.966} C_VEL
LIN {X 0,Y 578.49,Z 1019.905,A -85,B 0,C 180,E1 2065.497,E2 2065.497} C_VEL
LIN {X 0,Y 578.489,Z 1022.657,A -85,B 0,C 180,E1 2068.501,E2 2068.501} C_VEL
LIN {X 0,Y 578.434,Z 1021.627,A -85,B 0,C 180,E1 2073.001,E2 2073.001} C_VEL
LIN {X 0,Y 578.512,Z 1015.916,A -85,B 0,C 180,E1 2076.764,E2 2076.764} C_VEL
LIN {X 0,Y 578.563,Z 1005.776,A -85,B 0,C 180,E1 2080.556,E2 2080.556} C_VEL
LIN {X 0,Y 578.745,Z 988.612,A -85,B 0,C 180,E1 2084.8,E2 2084.8} C_VEL
LIN {X 0,Y 579.091,Z 965.906,A -85,B 0,C 180,E1 2088.846,E2 2088.846} C_VEL
LIN {X 0,Y 579.791,Z 937.988,A -85,B 0,C 180,E1 2092.62,E2 2092.62} C_VEL
LIN {X 0,Y 580.68,Z 905.14,A -85,B 0,C 180,E1 2096.055,E2 2096.055} C_VEL
LIN {X 0,Y 581.728,Z 869.474,A -85,B 0,C 180,E1 2098.947,E2 2098.947} C_VEL
LIN {X 0,Y 582.87,Z 830.017,A -85,B 0,C 180,E1 2101.366,E2 2101.366} C_VEL
LIN {X 0,Y 583.872,Z 789.965,A -85,B 0,C 180,E1 2103.127,E2 2103.127} C_VEL
LIN {X 0,Y 584.506,Z 750.861,A -85,B 0,C 180,E1 2104.251,E2 2104.251} C_VEL
LIN {X 0,Y 584.134,Z 705.116,A -85,B 0,C 180,E1 2105.044,E2 2105.044} C_VEL
LIN {X 0,Y 577.871,Z 691.44,A -85,B 0,C 180,E1 2105.69,E2 2105.69} C_VEL
LIN {X 0,Y 577.827,Z 691.44,A -85,B 0,C 180,E1 2110.926,E2 2110.926} C_VEL
LIN {X 0,Y 577.961,Z 691.44,A -85,B 0,C 180,E1 2117.071,E2 2117.071} C_VEL
LIN {X 0,Y 577.955,Z 691.44,A -85,B 0,C 180,E1 2122.95,E2 2122.95} C_VEL
LIN {X 0,Y 577.875,Z 691.44,A -85,B 0,C 180,E1 2128.399,E2 2128.399} C_VEL
LIN {X 0,Y 577.975,Z 691.44,A -85,B 0,C 180,E1 2133.555,E2 2133.555} C_VEL
LIN {X 0,Y 578.018,Z 691.44,A -85,B 0,C 180,E1 2138.486,E2 2138.486} C_VEL
LIN {X 0,Y 578.173,Z 691.44,A -85,B 0,C 180,E1 2143.257,E2 2143.257} C_VEL
LIN {X 0,Y 578.116,Z 691.44,A -85,B 0,C 180,E1 2149.434,E2 2149.434} C_VEL
LIN {X 0,Y 578.361,Z 691.44,A -85,B 0,C 180,E1 2154.155,E2 2154.155} C_VEL
LIN {X 0,Y 578.178,Z 691.44,A -85,B 0,C 180,E1 2159.996,E2 2159.996} C_VEL
LIN {X 0,Y 578.171,Z 691.44,A -85,B 0,C 180,E1 2164.502,E2 2164.502} C_VEL
LIN {X 0,Y 578.187,Z 691.44,A -85,B 0,C 180,E1 2169.035,E2 2169.035} C_VEL
LIN {X 0,Y 578.063,Z 691.44,A -85,B 0,C 180,E1 2174.275,E2 2174.275} C_VEL
LIN {X 0,Y 578.05,Z 691.44,A -85,B 0,C 180,E1 2179.901,E2 2179.901} C_VEL
LIN {X 0,Y 577.954,Z 691.44,A -85,B 0,C 180,E1 2184.774,E2 2184.774} C_VEL
LIN {X 0,Y 577.871,Z 691.44,A -85,B 0,C 180,E1 2190.158,E2 2190.158} C_VEL
LIN {X 0,Y 578.033,Z 691.44,A -85,B 0,C 180,E1 2195.178,E2 2195.178} C_VEL
LIN {X 0,Y 577.956,Z 691.44,A -85,B 0,C 180,E1 2200.903,E2 2200.903} C_VEL
LIN {X 0,Y 577.869,Z 691.44,A -85,B 0,C 180,E1 2207.178,E2 2207.178} C_VEL
LIN {X 0,Y 578.022,Z 691.44,A -85,B 0,C 180,E1 2212.953,E2 2212.953} C_VEL
LIN {X 0,Y 578.237,Z 691.44,A -85,B 0,C 180,E1 2214.711,E2 2214.711} C_VEL
LIN {X 0,Y 584.408,Z 705.512,A -85,B 0,C 180,E1 2215.393,E2 2215.393} C_VEL
LIN {X 0,Y 584.037,Z 747.203,A -85,B 0,C 180,E1 2216.396,E2 2216.396} C_VEL
LIN {X 0,Y 583.201,Z 788.037,A -85,B 0,C 180,E1 2217.993,E2 2217.993} C_VEL
LIN {X 0,Y 582.137,Z 827.783,A -85,B 0,C 180,E1 2220.214,E2 2220.214} C_VEL
LIN {X 0,Y 580.964,Z 865.163,A -85,B 0,C 180,E1 2223.01,E2 2223.01} C_VEL
LIN {X 0,Y 579.977,Z 898.922,A -85,B 0,C 180,E1 2226.294,E2 2226.294} C_VEL
LIN {X 0,Y 579.242,Z 927.976,A -85,B 0,C 180,E1 2229.935,E2 2229.935} C_VEL
LIN {X 0,Y 578.716,Z 952.067,A -85,B 0,C 180,E1 2233.86,E2 2233.86} C_VEL
LIN {X 0,Y 578.474,Z 970.487,A -85,B 0,C 180,E1 2237.913,E2 2237.913} C_VEL
LIN {X 0,Y 578.412,Z 982.517,A -85,B 0,C 180,E1 2241.722,E2 2241.722} C_VEL
LIN {X 0,Y 578.332,Z 989.967,A -85,B 0,C 180,E1 2245.495,E2 2245.495} C_VEL
LIN {X 0,Y 578.327,Z 992.676,A -85,B 0,C 180,E1 2248.5,E2 2248.5} C_VEL
LIN {X 0,Y 578.427,Z 992.63,A -85,B 0,C 180,E1 2251.5,E2 2251.5} C_VEL
LIN {X 0,Y 578.453,Z 987.312,A -85,B 0,C 180,E1 2256.046,E2 2256.046} C_VEL
LIN {X 0,Y 578.531,Z 976.846,A -85,B 0,C 180,E1 2260.175,E2 2260.175} C_VEL
LIN {X 0,Y 578.627,Z 961.716,A -85,B 0,C 180,E1 2264.077,E2 2264.077} C_VEL
LIN {X 0,Y 578.963,Z 941.665,A -85,B 0,C 180,E1 2267.872,E2 2267.872} C_VEL
LIN {X 0,Y 579.564,Z 915.599,A -85,B 0,C 180,E1 2271.634,E2 2271.634} C_VEL
LIN {X 0,Y 580.37,Z 885.865,A -85,B 0,C 180,E1 2274.98,E2 2274.98} C_VEL
LIN {X 0,Y 581.392,Z 851.097,A -85,B 0,C 180,E1 2278.038,E2 2278.038} C_VEL
LIN {X 0,Y 582.474,Z 814.413,A -85,B 0,C 180,E1 2280.524,E2 2280.524} C_VEL
LIN {X 0,Y 583.548,Z 772.475,A -85,B 0,C 180,E1 2282.605,E2 2282.605} C_VEL
LIN {X 0,Y 584.358,Z 731.304,A -85,B 0,C 180,E1 2283.964,E2 2283.964} C_VEL
LIN {X 0,Y 583.87,Z 704.642,A -85,B 0,C 180,E1 2284.569,E2 2284.569} C_VEL
LIN {X 0,Y 577.898,Z 691.44,A -85,B 0,C 180,E1 2285.197,E2 2285.197} C_VEL
LIN {X 0,Y 577.81,Z 691.44,A -85,B 0,C 180,E1 2290.927,E2 2290.927} C_VEL
LIN {X 0,Y 577.969,Z 691.44,A -85,B 0,C 180,E1 2297.082,E2 2297.082} C_VEL
LIN {X 0,Y 577.927,Z 691.44,A -85,B 0,C 180,E1 2302.957,E2 2302.957} C_VEL
LIN {X 0,Y 577.878,Z 691.44,A -85,B 0,C 180,E1 2308.407,E2 2308.407} C_VEL
LIN {X 0,Y 578,Z 691.44,A -85,B 0,C 180,E1 2313.564,E2 2313.564} C_VEL
LIN {X 0,Y 578.048,Z 691.44,A -85,B 0,C 180,E1 2318.495,E2 2318.495} C_VEL
LIN {X 0,Y 578.12,Z 691.44,A -85,B 0,C 180,E1 2323.263,E2 2323.263} C_VEL
LIN {X 0,Y 578.185,Z 691.44,A -85,B 0,C 180,E1 2327.913,E2 2327.913} C_VEL
LIN {X 0,Y 578.169,Z 691.44,A -85,B 0,C 180,E1 2332.481,E2 2332.481} C_VEL
LIN {X 0,Y 578.286,Z 691.44,A -85,B 0,C 180,E1 2337.002,E2 2337.002} C_VEL
LIN {X 0,Y 578.414,Z 691.44,A -85,B 0,C 180,E1 2341.503,E2 2341.503} C_VEL
LIN {X 0,Y 578.367,Z 691.44,A -85,B 0,C 180,E1 2346.014,E2 2346.014} C_VEL
LIN {X 0,Y 578.03,Z 691.44,A -85,B 0,C 180,E1 2347.593,E2 2347.593} C_VEL
LIN {X 0,Y 574.137,Z 691.44,A -85,B 0,C 180,E1 2349.286,E2 2349.286} C_VEL
LIN {X 0,Y 570.211,Z 691.44,A -85,B 0,C 180,E1 2351,E2 2351} C_VEL
LIN {X 0,Y 570.07,Z 691.44,A -85,B 0,C 180,E1 2357.032,E2 2357.032} C_VEL
LIN {X 0,Y 570.11,Z 691.44,A -85,B 0,C 180,E1 2361.828,E2 2361.828} C_VEL
LIN {X 0,Y 570.054,Z 691.44,A -85,B 0,C 180,E1 2366.842,E2 2366.842} C_VEL
LIN {X 0,Y 569.916,Z 691.44,A -85,B 0,C 180,E1 2372.095,E2 2372.095} C_VEL
LIN {X 0,Y 570.044,Z 691.44,A -85,B 0,C 180,E1 2377.653,E2 2377.653} C_VEL
LIN {X 0,Y 569.956,Z 691.44,A -85,B 0,C 180,E1 2383.682,E2 2383.682} C_VEL
LIN {X 0,Y 569.849,Z 691.44,A -85,B 0,C 180,E1 2388.376,E2 2388.376} C_VEL
LIN {X 0,Y 569.942,Z 692.197,A -85,B 0,C 180,E1 2393.751,E2 2393.751} C_VEL
LIN {X 0,Y 578.126,Z 709.122,A -85,B 0,C 180,E1 2394.597,E2 2394.597} C_VEL
LIN {X 0,Y 577.709,Z 759.852,A -85,B 0,C 180,E1 2395.503,E2 2395.503} C_VEL
LIN {X 0,Y 576.81,Z 801.651,A -85,B 0,C 180,E1 2396.887,E2 2396.887} C_VEL
LIN {X 0,Y 575.492,Z 842.698,A -85,B 0,C 180,E1 2398.919,E2 2398.919} C_VEL
LIN {X 0,Y 574.23,Z 880.694,A -85,B 0,C 180,E1 2401.503,E2 2401.503} C_VEL
LIN {X 0,Y 572.936,Z 915.382,A -85,B 0,C 180,E1 2404.579,E2 2404.579} C_VEL
LIN {X 0,Y 571.883,Z 945.791,A -85,B 0,C 180,E1 2408.039,E2 2408.039} C_VEL
LIN {X 0,Y 571.164,Z 971.308,A -85,B 0,C 180,E1 2411.771,E2 2411.771} C_VEL
LIN {X 0,Y 570.778,Z 990.971,A -85,B 0,C 180,E1 2415.513,E2 2415.513} C_VEL
LIN {X 0,Y 570.562,Z 1005.777,A -85,B 0,C 180,E1 2419.295,E2 2419.295} C_VEL
LIN {X 0,Y 570.471,Z 1015.917,A -85,B 0,C 180,E1 2423.141,E2 2423.141} C_VEL
LIN {X 0,Y 570.435,Z 1021.628,A -85,B 0,C 180,E1 2426.957,E2 2426.957} C_VEL
LIN {X 0,Y 570.442,Z 1023,A -85,B 0,C 180,E1 2430,E2 2430} C_VEL
LIN {X 0,Y 570.526,Z 1021.627,A -85,B 0,C 180,E1 2433.043,E2 2433.043} C_VEL
LIN {X 0,Y 570.605,Z 1015.916,A -85,B 0,C 180,E1 2436.858,E2 2436.858} C_VEL
LIN {X 0,Y 570.658,Z 1004.743,A -85,B 0,C 180,E1 2441.002,E2 2441.002} C_VEL
LIN {X 0,Y 570.926,Z 988.312,A -85,B 0,C 180,E1 2445.068,E2 2445.068} C_VEL
LIN {X 0,Y 571.343,Z 965.117,A -85,B 0,C 180,E1 2449.232,E2 2449.232} C_VEL
LIN {X 0,Y 572.195,Z 937.172,A -85,B 0,C 180,E1 2453.033,E2 2453.033} C_VEL
LIN {X 0,Y 573.325,Z 904.368,A -85,B 0,C 180,E1 2456.486,E2 2456.486} C_VEL
LIN {X 0,Y 574.641,Z 868.311,A -85,B 0,C 180,E1 2459.421,E2 2459.421} C_VEL
LIN {X 0,Y 575.988,Z 829.927,A -85,B 0,C 180,E1 2461.789,E2 2461.789} C_VEL
LIN {X 0,Y 577.213,Z 789.962,A -85,B 0,C 180,E1 2463.559,E2 2463.559} C_VEL
LIN {X 0,Y 577.963,Z 751.174,A -85,B 0,C 180,E1 2464.686,E2 2464.686} C_VEL
LIN {X 0,Y 577.677,Z 707.927,A -85,B 0,C 180,E1 2465.453,E2 2465.453} C_VEL
LIN {X 0,Y 569.933,Z 691.44,A -85,B 0,C 180,E1 2466.281,E2 2466.281} C_VEL
LIN {X 0,Y 569.849,Z 691.44,A -85,B 0,C 180,E1 2471.934,E2 2471.934} C_VEL
LIN {X 0,Y 569.967,Z 691.44,A -85,B 0,C 180,E1 2478.057,E2 2478.057} C_VEL
LIN {X 0,Y 569.988,Z 691.44,A -85,B 0,C 180,E1 2484.241,E2 2484.241} C_VEL
LIN {X 0,Y 569.992,Z 691.44,A -85,B 0,C 180,E1 2489.689,E2 2489.689} C_VEL
LIN {X 0,Y 570.111,Z 691.44,A -85,B 0,C 180,E1 2494.854,E2 2494.854} C_VEL
LIN {X 0,Y 570.161,Z 691.44,A -85,B 0,C 180,E1 2499.804,E2 2499.804} C_VEL
LIN {X 0,Y 570.002,Z 691.44,A -85,B 0,C 180,E1 2504.594,E2 2504.594} C_VEL
LIN {X 0,Y 570.106,Z 691.44,A -85,B 0,C 180,E1 2510.829,E2 2510.829} C_VEL
LIN {X 0,Y 570.231,Z 691.44,A -85,B 0,C 180,E1 2515.428,E2 2515.428} C_VEL
LIN {X 0,Y 570.291,Z 691.44,A -85,B 0,C 180,E1 2519.996,E2 2519.996} C_VEL
LIN {X 0,Y 570.274,Z 691.44,A -85,B 0,C 180,E1 2524.564,E2 2524.564} C_VEL
LIN {X 0,Y 570.255,Z 691.44,A -85,B 0,C 180,E1 2529.162,E2 2529.162} C_VEL
LIN {X 0,Y 570.268,Z 691.44,A -85,B 0,C 180,E1 2533.819,E2 2533.819} C_VEL
LIN {X 0,Y 570.219,Z 691.44,A -85,B 0,C 180,E1 2538.574,E2 2538.574} C_VEL
LIN {X 0,Y 570.132,Z 691.44,A -85,B 0,C 180,E1 2543.468,E2 2543.468} C_VEL
LIN {X 0,Y 570.014,Z 691.44,A -85,B 0,C 180,E1 2548.77,E2 2548.77} C_VEL
LIN {X 0,Y 570.13,Z 691.44,A -85,B 0,C 180,E1 2554.587,E2 2554.587} C_VEL
LIN {X 0,Y 569.995,Z 691.44,A -85,B 0,C 180,E1 2559.616,E2 2559.616} C_VEL
LIN {X 0,Y 569.801,Z 691.44,A -85,B 0,C 180,E1 2565.831,E2 2565.831} C_VEL
LIN {X 0,Y 570.021,Z 691.44,A -85,B 0,C 180,E1 2570.395,E2 2570.395} C_VEL
LIN {X 0,Y 570.23,Z 691.44,A -85,B 0,C 180,E1 2574.15,E2 2574.15} C_VEL
LIN {X 0,Y 578.021,Z 709.583,A -85,B 0,C 180,E1 2575.027,E2 2575.027} C_VEL
LIN {X 0,Y 577.359,Z 749.795,A -85,B 0,C 180,E1 2576.045,E2 2576.045} C_VEL
LIN {X 0,Y 576.341,Z 788.361,A -85,B 0,C 180,E1 2577.584,E2 2577.584} C_VEL
LIN {X 0,Y 575.029,Z 828.214,A -85,B 0,C 180,E1 2579.838,E2 2579.838} C_VEL
LIN {X 0,Y 573.612,Z 866.238,A -85,B 0,C 180,E1 2582.732,E2 2582.732} C_VEL
LIN {X 0,Y 572.444,Z 899.267,A -85,B 0,C 180,E1 2586.004,E2 2586.004} C_VEL
LIN {X 0,Y 571.528,Z 927.973,A -85,B 0,C 180,E1 2589.653,E2 2589.653} C_VEL
LIN {X 0,Y 570.932,Z 952.065,A -85,B 0,C 180,E1 2593.634,E2 2593.634} C_VEL
LIN {X 0,Y 570.632,Z 970.484,A -85,B 0,C 180,E1 2597.744,E2 2597.744} C_VEL
LIN {X 0,Y 570.53,Z 982.515,A -85,B 0,C 180,E1 2601.607,E2 2601.607} C_VEL
LIN {X 0,Y 570.462,Z 989.966,A -85,B 0,C 180,E1 2605.433,E2 2605.433} C_VEL
LIN {X 0,Y 570.438,Z 992.676,A -85,B 0,C 180,E1 2608.479,E2 2608.479} C_VEL
LIN {X 0,Y 570.527,Z 992.631,A -85,B 0,C 180,E1 2611.52,E2 2611.52} C_VEL
LIN {X 0,Y 570.573,Z 987.389,A -85,B 0,C 180,E1 2616.093,E2 2616.093} C_VEL
LIN {X 0,Y 570.643,Z 976.848,A -85,B 0,C 180,E1 2620.317,E2 2620.317} C_VEL
LIN {X 0,Y 570.77,Z 960.683,A -85,B 0,C 180,E1 2624.506,E2 2624.506} C_VEL
LIN {X 0,Y 571.211,Z 940.986,A -85,B 0,C 180,E1 2628.236,E2 2628.236} C_VEL
LIN {X 0,Y 571.894,Z 915.28,A -85,B 0,C 180,E1 2631.981,E2 2631.981} C_VEL
LIN {X 0,Y 572.973,Z 884.812,A -85,B 0,C 180,E1 2635.432,E2 2635.432} C_VEL
LIN {X 0,Y 574.221,Z 850.079,A -85,B 0,C 180,E1 2638.5,E2 2638.5} C_VEL
LIN {X 0,Y 575.534,Z 812.963,A -85,B 0,C 180,E1 2641.018,E2 2641.018} C_VEL
LIN {X 0,Y 576.804,Z 771.741,A -85,B 0,C 180,E1 2643.065,E2 2643.065} C_VEL
LIN {X 0,Y 577.798,Z 730.856,A -85,B 0,C 180,E1 2644.417,E2 2644.417} C_VEL
LIN {X 0,Y 577.419,Z 707.676,A -85,B 0,C 180,E1 2644.958,E2 2644.958} C_VEL
LIN {X 0,Y 569.949,Z 691.44,A -85,B 0,C 180,E1 2645.763,E2 2645.763} C_VEL
LIN {X 0,Y 569.847,Z 691.44,A -85,B 0,C 180,E1 2651.624,E2 2651.624} C_VEL
LIN {X 0,Y 569.969,Z 691.44,A -85,B 0,C 180,E1 2656.329,E2 2656.329} C_VEL
LIN {X 0,Y 570.009,Z 691.44,A -85,B 0,C 180,E1 2662.354,E2 2662.354} C_VEL
LIN {X 0,Y 569.965,Z 691.44,A -85,B 0,C 180,E1 2668.218,E2 2668.218} C_VEL
LIN {X 0,Y 570.13,Z 691.44,A -85,B 0,C 180,E1 2674.545,E2 2674.545} C_VEL
LIN {X 0,Y 570.204,Z 691.44,A -85,B 0,C 180,E1 2679.813,E2 2679.813} C_VEL
LIN {X 0,Y 570.393,Z 691.44,A -85,B 0,C 180,E1 2686.184,E2 2686.184} C_VEL
LIN {X 0,Y 570.261,Z 691.44,A -85,B 0,C 180,E1 2692.376,E2 2692.376} C_VEL
LIN {X 0,Y 570.378,Z 691.44,A -85,B 0,C 180,E1 2696.961,E2 2696.961} C_VEL
LIN {X 0,Y 570.516,Z 691.44,A -85,B 0,C 180,E1 2701.524,E2 2701.524} C_VEL
LIN {X 0,Y 570.435,Z 691.44,A -85,B 0,C 180,E1 2706.097,E2 2706.097} C_VEL
LIN {X 0,Y 570.211,Z 691.44,A -85,B 0,C 180,E1 2711,E2 2711} C_VEL
LIN {X 0,Y 566.167,Z 691.44,A -85,B 0,C 180,E1 2712.713,E2 2712.713} C_VEL
LIN {X 0,Y 562.196,Z 691.44,A -85,B 0,C 180,E1 2714.449,E2 2714.449} C_VEL
LIN {X 0,Y 562.23,Z 691.44,A -85,B 0,C 180,E1 2720.494,E2 2720.494} C_VEL
LIN {X 0,Y 562.227,Z 691.44,A -85,B 0,C 180,E1 2725.524,E2 2725.524} C_VEL
LIN {X 0,Y 562.038,Z 691.44,A -85,B 0,C 180,E1 2730.786,E2 2730.786} C_VEL
LIN {X 0,Y 562.093,Z 691.44,A -85,B 0,C 180,E1 2736.341,E2 2736.341} C_VEL
LIN {X 0,Y 562.029,Z 691.44,A -85,B 0,C 180,E1 2742.335,E2 2742.335} C_VEL
LIN {X 0,Y 561.923,Z 691.44,A -85,B 0,C 180,E1 2747.654,E2 2747.654} C_VEL
LIN {X 0,Y 562.013,Z 691.44,A -85,B 0,C 180,E1 2753.12,E2 2753.12} C_VEL
LIN {X 0,Y 571.689,Z 713.019,A -85,B 0,C 180,E1 2754.196,E2 2754.196} C_VEL
LIN {X 0,Y 571.127,Z 761.273,A -85,B 0,C 180,E1 2755.09,E2 2755.09} C_VEL
LIN {X 0,Y 570.062,Z 803.091,A -85,B 0,C 180,E1 2756.504,E2 2756.504} C_VEL
LIN {X 0,Y 568.48,Z 845.403,A -85,B 0,C 180,E1 2758.656,E2 2758.656} C_VEL
LIN {X 0,Y 566.882,Z 884.015,A -85,B 0,C 180,E1 2761.366,E2 2761.366} C_VEL
LIN {X 0,Y 565.334,Z 919.343,A -85,B 0,C 180,E1 2764.627,E2 2764.627} C_VEL
LIN {X 0,Y 564.217,Z 948.918,A -85,B 0,C 180,E1 2768.14,E2 2768.14} C_VEL
LIN {X 0,Y 563.376,Z 974.542,A -85,B 0,C 180,E1 2772.061,E2 2772.061} C_VEL
LIN {X 0,Y 562.938,Z 995.671,A -85,B 0,C 180,E1 2776.389,E2 2776.389} C_VEL
LIN {X 0,Y 562.764,Z 1010.44,A -85,B 0,C 180,E1 2780.711,E2 2780.711} C_VEL
LIN {X 0,Y 562.722,Z 1019.905,A -85,B 0,C 180,E1 2785.37,E2 2785.37} C_VEL
LIN {X 0,Y 562.684,Z 1022.657,A -85,B 0,C 180,E1 2788.458,E2 2788.458} C_VEL
LIN {X 0,Y 562.619,Z 1021.627,A -85,B 0,C 180,E1 2793.086,E2 2793.086} C_VEL
LIN {X 0,Y 562.728,Z 1015.916,A -85,B 0,C 180,E1 2796.955,E2 2796.955} C_VEL
LIN {X 0,Y 562.765,Z 1004.743,A -85,B 0,C 180,E1 2801.159,E2 2801.159} C_VEL
LIN {X 0,Y 563.087,Z 988.233,A -85,B 0,C 180,E1 2805.299,E2 2805.299} C_VEL
LIN {X 0,Y 563.593,Z 965.92,A -85,B 0,C 180,E1 2809.382,E2 2809.382} C_VEL
LIN {X 0,Y 564.632,Z 937.677,A -85,B 0,C 180,E1 2813.299,E2 2813.299} C_VEL
LIN {X 0,Y 565.937,Z 905.398,A -85,B 0,C 180,E1 2816.763,E2 2816.763} C_VEL
LIN {X 0,Y 567.493,Z 870.269,A -85,B 0,C 180,E1 2819.687,E2 2819.687} C_VEL
LIN {X 0,Y 569.1,Z 830.246,A -85,B 0,C 180,E1 2822.203,E2 2822.203} C_VEL
LIN {X 0,Y 570.528,Z 789.989,A -85,B 0,C 180,E1 2824.004,E2 2824.004} C_VEL
LIN {X 0,Y 571.441,Z 751.595,A -85,B 0,C 180,E1 2825.13,E2 2825.13} C_VEL
LIN {X 0,Y 571.045,Z 710.391,A -85,B 0,C 180,E1 2825.89,E2 2825.89} C_VEL
LIN {X 0,Y 562.024,Z 691.44,A -85,B 0,C 180,E1 2826.879,E2 2826.879} C_VEL
LIN {X 0,Y 561.929,Z 691.44,A -85,B 0,C 180,E1 2832.347,E2 2832.347} C_VEL
LIN {X 0,Y 562.033,Z 691.44,A -85,B 0,C 180,E1 2837.666,E2 2837.666} C_VEL
LIN {X 0,Y 562.091,Z 691.44,A -85,B 0,C 180,E1 2843.659,E2 2843.659} C_VEL
LIN {X 0,Y 562.078,Z 691.44,A -85,B 0,C 180,E1 2849.542,E2 2849.542} C_VEL
LIN {X 0,Y 562.187,Z 691.44,A -85,B 0,C 180,E1 2854.474,E2 2854.474} C_VEL
LIN {X 0,Y 562.247,Z 691.44,A -85,B 0,C 180,E1 2860.48,E2 2860.48} C_VEL
LIN {X 0,Y 562.11,Z 691.44,A -85,B 0,C 180,E1 2864.372,E2 2864.372} C_VEL
LIN {X 0,Y 562.224,Z 691.44,A -85,B 0,C 180,E1 2870.699,E2 2870.699} C_VEL
LIN {X 0,Y 562.333,Z 691.44,A -85,B 0,C 180,E1 2875.364,E2 2875.364} C_VEL
LIN {X 0,Y 562.391,Z 691.44,A -85,B 0,C 180,E1 2879.996,E2 2879.996} C_VEL
LIN {X 0,Y 562.311,Z 691.44,A -85,B 0,C 180,E1 2884.95,E2 2884.95} C_VEL
LIN {X 0,Y 562.345,Z 691.44,A -85,B 0,C 180,E1 2889.292,E2 2889.292} C_VEL
LIN {X 0,Y 562.306,Z 691.44,A -85,B 0,C 180,E1 2894.222,E2 2894.222} C_VEL
LIN {X 0,Y 562.223,Z 691.44,A -85,B 0,C 180,E1 2899.513,E2 2899.513} C_VEL
LIN {X 0,Y 562.104,Z 691.44,A -85,B 0,C 180,E1 2905.522,E2 2905.522} C_VEL
LIN {X 0,Y 562.09,Z 691.44,A -85,B 0,C 180,E1 2910.775,E2 2910.775} C_VEL
LIN {X 0,Y 562.164,Z 691.44,A -85,B 0,C 180,E1 2916.326,E2 2916.326} C_VEL
LIN {X 0,Y 561.974,Z 691.44,A -85,B 0,C 180,E1 2922.33,E2 2922.33} C_VEL
LIN {X 0,Y 561.975,Z 691.44,A -85,B 0,C 180,E1 2927.658,E2 2927.658} C_VEL
LIN {X 0,Y 562.263,Z 691.44,A -85,B 0,C 180,E1 2933.554,E2 2933.554} C_VEL
LIN {X 0,Y 571.53,Z 711.471,A -85,B 0,C 180,E1 2934.606,E2 2934.606} C_VEL
LIN {X 0,Y 570.71,Z 751.739,A -85,B 0,C 180,E1 2935.663,E2 2935.663} C_VEL
LIN {X 0,Y 569.464,Z 790.671,A -85,B 0,C 180,E1 2937.266,E2 2937.266} C_VEL
LIN {X 0,Y 567.918,Z 829.221,A -85,B 0,C 180,E1 2939.493,E2 2939.493} C_VEL
LIN {X 0,Y 566.301,Z 866.817,A -85,B 0,C 180,E1 2942.405,E2 2942.405} C_VEL
LIN {X 0,Y 564.91,Z 900.362,A -85,B 0,C 180,E1 2945.795,E2 2945.795} C_VEL
LIN {X 0,Y 563.884,Z 927.971,A -85,B 0,C 180,E1 2949.364,E2 2949.364} C_VEL
LIN {X 0,Y 563.154,Z 952.063,A -85,B 0,C 180,E1 2953.401,E2 2953.401} C_VEL
LIN {X 0,Y 562.764,Z 970.48,A -85,B 0,C 180,E1 2957.57,E2 2957.57} C_VEL
LIN {X 0,Y 562.642,Z 982.514,A -85,B 0,C 180,E1 2961.488,E2 2961.488} C_VEL
LIN {X 0,Y 562.562,Z 989.965,A -85,B 0,C 180,E1 2965.368,E2 2965.368} C_VEL
LIN {X 0,Y 562.538,Z 992.676,A -85,B 0,C 180,E1 2968.457,E2 2968.457} C_VEL
LIN {X 0,Y 562.621,Z 992.631,A -85,B 0,C 180,E1 2971.542,E2 2971.542} C_VEL
LIN {X 0,Y 562.67,Z 987.391,A -85,B 0,C 180,E1 2976.179,E2 2976.179} C_VEL
LIN {X 0,Y 562.75,Z 976.851,A -85,B 0,C 180,E1 2980.463,E2 2980.463} C_VEL
LIN {X 0,Y 562.94,Z 960.802,A -85,B 0,C 180,E1 2984.687,E2 2984.687} C_VEL
LIN {X 0,Y 563.454,Z 940.807,A -85,B 0,C 180,E1 2988.526,E2 2988.526} C_VEL
LIN {X 0,Y 564.289,Z 915.598,A -85,B 0,C 180,E1 2992.252,E2 2992.252} C_VEL
LIN {X 0,Y 565.555,Z 885.485,A -85,B 0,C 180,E1 2995.722,E2 2995.722} C_VEL
LIN {X 0,Y 567.068,Z 850.438,A -85,B 0,C 180,E1 2998.866,E2 2998.866} C_VEL
LIN {X 0,Y 568.58,Z 813.351,A -85,B 0,C 180,E1 3001.419,E2 3001.419} C_VEL
LIN {X 0,Y 570.045,Z 773.66,A -85,B 0,C 180,E1 3003.426,E2 3003.426} C_VEL
LIN {X 0,Y 571.153,Z 733.856,A -85,B 0,C 180,E1 3004.787,E2 3004.787} C_VEL
LIN {X 0,Y 571.145,Z 710.73,A -85,B 0,C 180,E1 3005.345,E2 3005.345} C_VEL
LIN {X 0,Y 562.108,Z 692.779,A -85,B 0,C 180,E1 3006.314,E2 3006.314} C_VEL
LIN {X 0,Y 561.998,Z 691.44,A -85,B 0,C 180,E1 3006.349,E2 3006.349} C_VEL
LIN {X 0,Y 561.925,Z 691.44,A -85,B 0,C 180,E1 3012.346,E2 3012.346} C_VEL
LIN {X 0,Y 562.039,Z 691.44,A -85,B 0,C 180,E1 3017.676,E2 3017.676} C_VEL
LIN {X 0,Y 562.1,Z 691.44,A -85,B 0,C 180,E1 3023.909,E2 3023.909} C_VEL
LIN {X 0,Y 562.09,Z 691.44,A -85,B 0,C 180,E1 3029.538,E2 3029.538} C_VEL
LIN {X 0,Y 562.249,Z 691.44,A -85,B 0,C 180,E1 3034.485,E2 3034.485} C_VEL
LIN {X 0,Y 562.28,Z 691.44,A -85,B 0,C 180,E1 3040.469,E2 3040.469} C_VEL
LIN {X 0,Y 562.448,Z 691.44,A -85,B 0,C 180,E1 3045.985,E2 3045.985} C_VEL
LIN {X 0,Y 562.359,Z 691.44,A -85,B 0,C 180,E1 3052.268,E2 3052.268} C_VEL
LIN {X 0,Y 562.47,Z 691.44,A -85,B 0,C 180,E1 3056.918,E2 3056.918} C_VEL
LIN {X 0,Y 562.605,Z 691.44,A -85,B 0,C 180,E1 3061.546,E2 3061.546} C_VEL
LIN {X 0,Y 562.523,Z 691.44,A -85,B 0,C 180,E1 3066.184,E2 3066.184} C_VEL
LIN {X 0,Y 562.226,Z 691.44,A -85,B 0,C 180,E1 3072.443,E2 3072.443} C_VEL
LIN {X 0,Y 562.196,Z 691.44,A -85,B 0,C 180,E1 3074.449,E2 3074.449} C_VEL
LIN {X 0,Y 558.211,Z 691.44,A -85,B 0,C 180,E1 3076.191,E2 3076.191} C_VEL
LIN {X 0,Y 554.208,Z 691.44,A -85,B 0,C 180,E1 3077.958,E2 3077.958} C_VEL
LIN {X 0,Y 554.251,Z 691.44,A -85,B 0,C 180,E1 3082.486,E2 3082.486} C_VEL
LIN {X 0,Y 554.154,Z 691.44,A -85,B 0,C 180,E1 3087.677,E2 3087.677} C_VEL
LIN {X 0,Y 554.044,Z 691.44,A -85,B 0,C 180,E1 3093.13,E2 3093.13} C_VEL
LIN {X 0,Y 554.133,Z 691.44,A -85,B 0,C 180,E1 3098.934,E2 3098.934} C_VEL
LIN {X 0,Y 554.129,Z 691.44,A -85,B 0,C 180,E1 3104.732,E2 3104.732} C_VEL
LIN {X 0,Y 554.012,Z 691.44,A -85,B 0,C 180,E1 3111.055,E2 3111.055} C_VEL
LIN {X 0,Y 554.106,Z 691.464,A -85,B 0,C 180,E1 3112.53,E2 3112.53} C_VEL
LIN {X 0,Y 560.416,Z 705.308,A -85,B 0,C 180,E1 3113.24,E2 3113.24} C_VEL
LIN {X 0,Y 565.197,Z 714.413,A -85,B 0,C 180,E1 3113.742,E2 3113.742} C_VEL
LIN {X 0,Y 564.589,Z 762.511,A -85,B 0,C 180,E1 3114.663,E2 3114.663} C_VEL
LIN {X 0,Y 563.352,Z 803.483,A -85,B 0,C 180,E1 3116.069,E2 3116.069} C_VEL
LIN {X 0,Y 561.544,Z 845.399,A -85,B 0,C 180,E1 3118.224,E2 3118.224} C_VEL
LIN {X 0,Y 559.72,Z 884.011,A -85,B 0,C 180,E1 3120.965,E2 3120.965} C_VEL
LIN {X 0,Y 557.919,Z 919.342,A -85,B 0,C 180,E1 3124.265,E2 3124.265} C_VEL
LIN {X 0,Y 556.562,Z 948.571,A -85,B 0,C 180,E1 3127.774,E2 3127.774} C_VEL
LIN {X 0,Y 555.621,Z 974.199,A -85,B 0,C 180,E1 3131.738,E2 3131.738} C_VEL
LIN {X 0,Y 555.068,Z 993.99,A -85,B 0,C 180,E1 3135.789,E2 3135.789} C_VEL
LIN {X 0,Y 554.815,Z 1008.484,A -85,B 0,C 180,E1 3139.902,E2 3139.902} C_VEL
LIN {X 0,Y 554.718,Z 1017.479,A -85,B 0,C 180,E1 3143.732,E2 3143.732} C_VEL
LIN {X 0,Y 554.654,Z 1021.628,A -85,B 0,C 180,E1 3146.871,E2 3146.871} C_VEL
LIN {X 0,Y 554.643,Z 1023,A -85,B 0,C 180,E1 3150,E2 3150} C_VEL
LIN {X 0,Y 554.726,Z 1021.627,A -85,B 0,C 180,E1 3153.13,E2 3153.13} C_VEL
LIN {X 0,Y 554.84,Z 1015.916,A -85,B 0,C 180,E1 3157.054,E2 3157.054} C_VEL
LIN {X 0,Y 554.895,Z 1005.774,A -85,B 0,C 180,E1 3161.012,E2 3161.012} C_VEL
LIN {X 0,Y 555.237,Z 989.306,A -85,B 0,C 180,E1 3165.286,E2 3165.286} C_VEL
LIN {X 0,Y 555.869,Z 966.343,A -85,B 0,C 180,E1 3169.592,E2 3169.592} C_VEL
LIN {X 0,Y 557.101,Z 937.679,A -85,B 0,C 180,E1 3173.633,E2 3173.633} C_VEL
LIN {X 0,Y 558.651,Z 905.26,A -85,B 0,C 180,E1 3177.153,E2 3177.153} C_VEL
LIN {X 0,Y 560.47,Z 869.091,A -85,B 0,C 180,E1 3180.185,E2 3180.185} C_VEL
LIN {X 0,Y 562.252,Z 831.26,A -85,B 0,C 180,E1 3182.587,E2 3182.587} C_VEL
LIN {X 0,Y 563.854,Z 791.63,A -85,B 0,C 180,E1 3184.395,E2 3184.395} C_VEL
LIN {X 0,Y 564.913,Z 754.451,A -85,B 0,C 180,E1 3185.529,E2 3185.529} C_VEL
LIN {X 0,Y 564.788,Z 713.657,A -85,B 0,C 180,E1 3186.3,E2 3186.3} C_VEL
LIN {X 0,Y 554.227,Z 692.755,A -85,B 0,C 180,E1 3187.44,E2 3187.44} C_VEL
LIN {X 0,Y 554.122,Z 691.44,A -85,B 0,C 180,E1 3187.594,E2 3187.594} C_VEL
LIN {X 0,Y 554.054,Z 691.44,A -85,B 0,C 180,E1 3193.093,E2 3193.093} C_VEL
LIN {X 0,Y 554.116,Z 691.44,A -85,B 0,C 180,E1 3199.023,E2 3199.023} C_VEL
LIN {X 0,Y 554.092,Z 691.44,A -85,B 0,C 180,E1 3205.062,E2 3205.062} C_VEL
LIN {X 0,Y 554.126,Z 691.44,A -85,B 0,C 180,E1 3210.97,E2 3210.97} C_VEL
LIN {X 0,Y 554.223,Z 691.44,A -85,B 0,C 180,E1 3215.808,E2 3215.808} C_VEL
LIN {X 0,Y 554.357,Z 691.44,A -85,B 0,C 180,E1 3220.867,E2 3220.867} C_VEL
LIN {X 0,Y 554.031,Z 691.44,A -85,B 0,C 180,E1 3225.76,E2 3225.76} C_VEL
LIN {X 0,Y 554.313,Z 691.44,A -85,B 0,C 180,E1 3230.565,E2 3230.565} C_VEL
LIN {X 0,Y 554.457,Z 691.44,A -85,B 0,C 180,E1 3235.298,E2 3235.298} C_VEL
LIN {X 0,Y 554.49,Z 691.44,A -85,B 0,C 180,E1 3239.996,E2 3239.996} C_VEL
LIN {X 0,Y 554.468,Z 691.44,A -85,B 0,C 180,E1 3244.695,E2 3244.695} C_VEL
LIN {X 0,Y 554.32,Z 691.44,A -85,B 0,C 180,E1 3250.48,E2 3250.48} C_VEL
LIN {X 0,Y 554.273,Z 691.44,A -85,B 0,C 180,E1 3255.847,E2 3255.847} C_VEL
LIN {X 0,Y 554.273,Z 691.44,A -85,B 0,C 180,E1 3260.793,E2 3260.793} C_VEL
LIN {X 0,Y 554.164,Z 691.44,A -85,B 0,C 180,E1 3265.914,E2 3265.914} C_VEL
LIN {X 0,Y 554.153,Z 691.44,A -85,B 0,C 180,E1 3271.264,E2 3271.264} C_VEL
LIN {X 0,Y 554.164,Z 691.44,A -85,B 0,C 180,E1 3276.937,E2 3276.937} C_VEL
LIN {X 0,Y 554.073,Z 691.44,A -85,B 0,C 180,E1 3282.454,E2 3282.454} C_VEL
LIN {X 0,Y 554.114,Z 691.44,A -85,B 0,C 180,E1 3289.02,E2 3289.02} C_VEL
LIN {X 0,Y 554.347,Z 691.44,A -85,B 0,C 180,E1 3292.972,E2 3292.972} C_VEL
LIN {X 0,Y 560.484,Z 704.949,A -85,B 0,C 180,E1 3293.68,E2 3293.68} C_VEL
LIN {X 0,Y 565.036,Z 714.957,A -85,B 0,C 180,E1 3294.207,E2 3294.207} C_VEL
LIN {X 0,Y 564.073,Z 754.639,A -85,B 0,C 180,E1 3295.306,E2 3295.306} C_VEL
LIN {X 0,Y 562.601,Z 792.547,A -85,B 0,C 180,E1 3296.918,E2 3296.918} C_VEL
LIN {X 0,Y 560.871,Z 830.217,A -85,B 0,C 180,E1 3299.142,E2 3299.142} C_VEL
LIN {X 0,Y 559.036,Z 866.613,A -85,B 0,C 180,E1 3301.997,E2 3301.997} C_VEL
LIN {X 0,Y 557.444,Z 900.356,A -85,B 0,C 180,E1 3305.45,E2 3305.45} C_VEL
LIN {X 0,Y 556.17,Z 929.31,A -85,B 0,C 180,E1 3309.273,E2 3309.273} C_VEL
LIN {X 0,Y 555.339,Z 952.061,A -85,B 0,C 180,E1 3313.161,E2 3313.161} C_VEL
LIN {X 0,Y 554.925,Z 970.477,A -85,B 0,C 180,E1 3317.392,E2 3317.392} C_VEL
LIN {X 0,Y 554.749,Z 982.513,A -85,B 0,C 180,E1 3321.366,E2 3321.366} C_VEL
LIN {X 0,Y 554.673,Z 989.964,A -85,B 0,C 180,E1 3325.302,E2 3325.302} C_VEL
LIN {X 0,Y 554.638,Z 992.675,A -85,B 0,C 180,E1 3328.435,E2 3328.435} C_VEL
LIN {X 0,Y 554.716,Z 992.632,A -85,B 0,C 180,E1 3331.564,E2 3331.564} C_VEL
LIN {X 0,Y 554.756,Z 987.392,A -85,B 0,C 180,E1 3336.267,E2 3336.267} C_VEL
LIN {X 0,Y 554.876,Z 976.161,A -85,B 0,C 180,E1 3340.849,E2 3340.849} C_VEL
LIN {X 0,Y 555.106,Z 960.351,A -85,B 0,C 180,E1 3345.004,E2 3345.004} C_VEL
LIN {X 0,Y 555.697,Z 940.325,A -85,B 0,C 180,E1 3348.877,E2 3348.877} C_VEL
LIN {X 0,Y 556.712,Z 915.615,A -85,B 0,C 180,E1 3352.57,E2 3352.57} C_VEL
LIN {X 0,Y 558.194,Z 885.061,A -85,B 0,C 180,E1 3356.131,E2 3356.131} C_VEL
LIN {X 0,Y 559.906,Z 850.52,A -85,B 0,C 180,E1 3359.265,E2 3359.265} C_VEL
LIN {X 0,Y 561.704,Z 813.367,A -85,B 0,C 180,E1 3361.848,E2 3361.848} C_VEL
LIN {X 0,Y 563.414,Z 772.401,A -85,B 0,C 180,E1 3363.93,E2 3363.93} C_VEL
LIN {X 0,Y 564.735,Z 732.042,A -85,B 0,C 180,E1 3365.296,E2 3365.296} C_VEL
LIN {X 0,Y 564.457,Z 713.29,A -85,B 0,C 180,E1 3365.782,E2 3365.782} C_VEL
LIN {X 0,Y 554.141,Z 692.86,A -85,B 0,C 180,E1 3366.922,E2 3366.922} C_VEL
LIN {X 0,Y 554.008,Z 691.44,A -85,B 0,C 180,E1 3366.959,E2 3366.959} C_VEL
LIN {X 0,Y 554.044,Z 691.44,A -85,B 0,C 180,E1 3373.094,E2 3373.094} C_VEL
LIN {X 0,Y 554.111,Z 691.44,A -85,B 0,C 180,E1 3379.032,E2 3379.032} C_VEL
LIN {X 0,Y 554.072,Z 691.44,A -85,B 0,C 180,E1 3385.064,E2 3385.064} C_VEL
LIN {X 0,Y 554.153,Z 691.44,A -85,B 0,C 180,E1 3390.964,E2 3390.964} C_VEL
LIN {X 0,Y 554.255,Z 691.44,A -85,B 0,C 180,E1 3395.818,E2 3395.818} C_VEL
LIN {X 0,Y 554.369,Z 691.44,A -85,B 0,C 180,E1 3400.875,E2 3400.875} C_VEL
LIN {X 0,Y 554.529,Z 691.44,A -85,B 0,C 180,E1 3405.781,E2 3405.781} C_VEL
LIN {X 0,Y 554.447,Z 691.44,A -85,B 0,C 180,E1 3412.157,E2 3412.157} C_VEL
LIN {X 0,Y 554.584,Z 691.44,A -85,B 0,C 180,E1 3416.874,E2 3416.874} C_VEL
LIN {X 0,Y 554.694,Z 691.44,A -85,B 0,C 180,E1 3421.568,E2 3421.568} C_VEL
LIN {X 0,Y 554.592,Z 691.44,A -85,B 0,C 180,E1 3426.272,E2 3426.272} C_VEL
LIN {X 0,Y 554.305,Z 691.44,A -85,B 0,C 180,E1 3432.624,E2 3432.624} C_VEL
LIN {X 0,Y 554.208,Z 691.44,A -85,B 0,C 180,E1 3437.958,E2 3437.958} C_VEL
LIN {X 0,Y 550.299,Z 691.44,A -85,B 0,C 180,E1 3439.724,E2 3439.724} C_VEL
LIN {X 0,Y 546.325,Z 691.44,A -85,B 0,C 180,E1 3441.514,E2 3441.514} C_VEL
LIN {X 0,Y 546.306,Z 691.44,A -85,B 0,C 180,E1 3446.324,E2 3446.324} C_VEL
LIN {X 0,Y 546.136,Z 691.44,A -85,B 0,C 180,E1 3451.786,E2 3451.786} C_VEL
LIN {X 0,Y 546.213,Z 691.44,A -85,B 0,C 180,E1 3457.576,E2 3457.576} C_VEL
LIN {X 0,Y 546.208,Z 691.44,A -85,B 0,C 180,E1 3463.887,E2 3463.887} C_VEL
LIN {X 0,Y 546.098,Z 691.44,A -85,B 0,C 180,E1 3470.381,E2 3470.381} C_VEL
LIN {X 0,Y 546.137,Z 691.44,A -85,B 0,C 180,E1 3471.866,E2 3471.866} C_VEL
LIN {X 0,Y 552.82,Z 705.654,A -85,B 0,C 180,E1 3472.655,E2 3472.655} C_VEL
LIN {X 0,Y 558.754,Z 717.163,A -85,B 0,C 180,E1 3473.299,E2 3473.299} C_VEL
LIN {X 0,Y 558.094,Z 763.005,A -85,B 0,C 180,E1 3474.204,E2 3474.204} C_VEL
LIN {X 0,Y 556.689,Z 804.148,A -85,B 0,C 180,E1 3475.639,E2 3475.639} C_VEL
LIN {X 0,Y 554.716,Z 845.432,A -85,B 0,C 180,E1 3477.788,E2 3477.788} C_VEL
LIN {X 0,Y 552.523,Z 884.457,A -85,B 0,C 180,E1 3480.59,E2 3480.59} C_VEL
LIN {X 0,Y 550.55,Z 919.342,A -85,B 0,C 180,E1 3483.895,E2 3483.895} C_VEL
LIN {X 0,Y 548.905,Z 949.905,A -85,B 0,C 180,E1 3487.64,E2 3487.64} C_VEL
LIN {X 0,Y 547.84,Z 975.299,A -85,B 0,C 180,E1 3491.677,E2 3491.677} C_VEL
LIN {X 0,Y 547.212,Z 995.673,A -85,B 0,C 180,E1 3495.99,E2 3495.99} C_VEL
LIN {X 0,Y 546.982,Z 1010.44,A -85,B 0,C 180,E1 3500.44,E2 3500.44} C_VEL
LIN {X 0,Y 546.919,Z 1018.703,A -85,B 0,C 180,E1 3504.44,E2 3504.44} C_VEL
LIN {X 0,Y 546.872,Z 1022.657,A -85,B 0,C 180,E1 3508.414,E2 3508.414} C_VEL
LIN {X 0,Y 546.819,Z 1021.627,A -85,B 0,C 180,E1 3513.175,E2 3513.175} C_VEL
LIN {X 0,Y 546.944,Z 1015.916,A -85,B 0,C 180,E1 3517.156,E2 3517.156} C_VEL
LIN {X 0,Y 547.01,Z 1005.774,A -85,B 0,C 180,E1 3521.172,E2 3521.172} C_VEL
LIN {X 0,Y 547.407,Z 988.717,A -85,B 0,C 180,E1 3525.645,E2 3525.645} C_VEL
LIN {X 0,Y 548.226,Z 965.626,A -85,B 0,C 180,E1 3529.996,E2 3529.996} C_VEL
LIN {X 0,Y 549.594,Z 937.674,A -85,B 0,C 180,E1 3533.976,E2 3533.976} C_VEL
LIN {X 0,Y 551.378,Z 904.779,A -85,B 0,C 180,E1 3537.588,E2 3537.588} C_VEL
LIN {X 0,Y 553.435,Z 869.094,A -85,B 0,C 180,E1 3540.609,E2 3540.609} C_VEL
LIN {X 0,Y 555.473,Z 831.259,A -85,B 0,C 180,E1 3543.035,E2 3543.035} C_VEL
LIN {X 0,Y 557.267,Z 790.987,A -85,B 0,C 180,E1 3544.887,E2 3544.887} C_VEL
LIN {X 0,Y 558.482,Z 754.453,A -85,B 0,C 180,E1 3546.001,E2 3546.001} C_VEL
LIN {X 0,Y 558.353,Z 716.319,A -85,B 0,C 180,E1 3546.745,E2 3546.745} C_VEL
LIN {X 0,Y 546.149,Z 691.44,A -85,B 0,C 180,E1 3548.135,E2 3548.135} C_VEL
LIN {X 0,Y 546.132,Z 691.44,A -85,B 0,C 180,E1 3553.881,E2 3553.881} C_VEL
LIN {X 0,Y 546.186,Z 691.44,A -85,B 0,C 180,E1 3558.458,E2 3558.458} C_VEL
LIN {X 0,Y 546.132,Z 691.44,A -85,B 0,C 180,E1 3564.396,E2 3564.396} C_VEL
LIN {X 0,Y 546.145,Z 691.44,A -85,B 0,C 180,E1 3570.065,E2 3570.065} C_VEL
LIN {X 0,Y 546.298,Z 691.44,A -85,B 0,C 180,E1 3576.151,E2 3576.151} C_VEL
LIN {X 0,Y 546.459,Z 691.44,A -85,B 0,C 180,E1 3582.254,E2 3582.254} C_VEL
LIN {X 0,Y 546.383,Z 691.44,A -85,B 0,C 180,E1 3588.813,E2 3588.813} C_VEL
LIN {X 0,Y 546.57,Z 691.44,A -85,B 0,C 180,E1 3595.23,E2 3595.23} C_VEL
LIN {X 0,Y 546.59,Z 691.44,A -85,B 0,C 180,E1 3599.996,E2 3599.996} C_VEL
LIN {X 0,Y 546.586,Z 691.44,A -85,B 0,C 180,E1 3604.762,E2 3604.762} C_VEL
LIN {X 0,Y 546.499,Z 691.44,A -85,B 0,C 180,E1 3609.564,E2 3609.564} C_VEL
LIN {X 0,Y 546.481,Z 691.44,A -85,B 0,C 180,E1 3614.433,E2 3614.433} C_VEL
LIN {X 0,Y 546.404,Z 691.44,A -85,B 0,C 180,E1 3619.585,E2 3619.585} C_VEL
LIN {X 0,Y 546.302,Z 691.44,A -85,B 0,C 180,E1 3624.557,E2 3624.557} C_VEL
LIN {X 0,Y 546.219,Z 691.44,A -85,B 0,C 180,E1 3629.921,E2 3629.921} C_VEL
LIN {X 0,Y 546.282,Z 691.44,A -85,B 0,C 180,E1 3635.584,E2 3635.584} C_VEL
LIN {X 0,Y 546.144,Z 691.44,A -85,B 0,C 180,E1 3641.697,E2 3641.697} C_VEL
LIN {X 0,Y 546.155,Z 691.44,A -85,B 0,C 180,E1 3648.447,E2 3648.447} C_VEL
LIN {X 0,Y 546.339,Z 691.44,A -85,B 0,C 180,E1 3652.335,E2 3652.335} C_VEL
LIN {X 0,Y 552.946,Z 705.708,A -85,B 0,C 180,E1 3653.119,E2 3653.119} C_VEL
LIN {X 0,Y 558.534,Z 718.088,A -85,B 0,C 180,E1 3653.802,E2 3653.802} C_VEL
LIN {X 0,Y 557.428,Z 757.259,A -85,B 0,C 180,E1 3654.928,E2 3654.928} C_VEL
LIN {X 0,Y 555.62,Z 797.331,A -85,B 0,C 180,E1 3656.711,E2 3656.711} C_VEL
LIN {X 0,Y 553.642,Z 834.883,A -85,B 0,C 180,E1 3659.043,E2 3659.043} C_VEL
LIN {X 0,Y 551.653,Z 869.505,A -85,B 0,C 180,E1 3661.87,E2 3661.87} C_VEL
LIN {X 0,Y 549.868,Z 902.027,A -85,B 0,C 180,E1 3665.295,E2 3665.295} C_VEL
LIN {X 0,Y 548.515,Z 929.307,A -85,B 0,C 180,E1 3668.97,E2 3668.97} C_VEL
LIN {X 0,Y 547.577,Z 952.207,A -85,B 0,C 180,E1 3672.946,E2 3672.946} C_VEL
LIN {X 0,Y 547.065,Z 970.473,A -85,B 0,C 180,E1 3677.208,E2 3677.208} C_VEL
LIN {X 0,Y 546.86,Z 982.511,A -85,B 0,C 180,E1 3681.241,E2 3681.241} C_VEL
LIN {X 0,Y 546.786,Z 990.051,A -85,B 0,C 180,E1 3685.313,E2 3685.313} C_VEL
LIN {X 0,Y 546.738,Z 992.675,A -85,B 0,C 180,E1 3688.413,E2 3688.413} C_VEL
LIN {X 0,Y 546.81,Z 992.633,A -85,B 0,C 180,E1 3691.586,E2 3691.586} C_VEL
LIN {X 0,Y 546.871,Z 988.635,A -85,B 0,C 180,E1 3695.561,E2 3695.561} C_VEL
LIN {X 0,Y 547.003,Z 980.311,A -85,B 0,C 180,E1 3699.56,E2 3699.56} C_VEL
LIN {X 0,Y 547.238,Z 965.503,A -85,B 0,C 180,E1 3704.01,E2 3704.01} C_VEL
LIN {X 0,Y 547.863,Z 945.062,A -85,B 0,C 180,E1 3708.322,E2 3708.322} C_VEL
LIN {X 0,Y 548.924,Z 919.475,A -85,B 0,C 180,E1 3712.376,E2 3712.376} C_VEL
LIN {X 0,Y 550.718,Z 887.49,A -85,B 0,C 180,E1 3716.259,E2 3716.259} C_VEL
LIN {X 0,Y 552.705,Z 852.245,A -85,B 0,C 180,E1 3719.544,E2 3719.544} C_VEL
LIN {X 0,Y 554.79,Z 814.272,A -85,B 0,C 180,E1 3722.238,E2 3722.238} C_VEL
LIN {X 0,Y 556.764,Z 773.13,A -85,B 0,C 180,E1 3724.36,E2 3724.36} C_VEL
LIN {X 0,Y 558.202,Z 733.524,A -85,B 0,C 180,E1 3725.728,E2 3725.728} C_VEL
LIN {X 0,Y 558.019,Z 716.202,A -85,B 0,C 180,E1 3726.193,E2 3726.193} C_VEL
LIN {X 0,Y 546.339,Z 693.274,A -85,B 0,C 180,E1 3727.534,E2 3727.534} C_VEL
LIN {X 0,Y 546.103,Z 691.44,A -85,B 0,C 180,E1 3727.586,E2 3727.586} C_VEL
LIN {X 0,Y 546.126,Z 691.44,A -85,B 0,C 180,E1 3733.891,E2 3733.891} C_VEL
LIN {X 0,Y 546.179,Z 691.44,A -85,B 0,C 180,E1 3738.458,E2 3738.458} C_VEL
LIN {X 0,Y 546.109,Z 691.44,A -85,B 0,C 180,E1 3744.403,E2 3744.403} C_VEL
LIN {X 0,Y 546.167,Z 691.44,A -85,B 0,C 180,E1 3750.075,E2 3750.075} C_VEL
LIN {X 0,Y 546.328,Z 691.44,A -85,B 0,C 180,E1 3756.142,E2 3756.142} C_VEL
LIN {X 0,Y 546.427,Z 691.44,A -85,B 0,C 180,E1 3760.586,E2 3760.586} C_VEL
LIN {X 0,Y 546.642,Z 691.44,A -85,B 0,C 180,E1 3765.794,E2 3765.794} C_VEL
LIN {X 0,Y 546.535,Z 691.44,A -85,B 0,C 180,E1 3772.043,E2 3772.043} C_VEL
LIN {X 0,Y 546.675,Z 691.44,A -85,B 0,C 180,E1 3776.829,E2 3776.829} C_VEL
LIN {X 0,Y 546.784,Z 691.44,A -85,B 0,C 180,E1 3781.59,E2 3781.59} C_VEL
LIN {X 0,Y 546.662,Z 691.44,A -85,B 0,C 180,E1 3786.364,E2 3786.364} C_VEL
LIN {X 0,Y 546.386,Z 691.44,A -85,B 0,C 180,E1 3792.81,E2 3792.81} C_VEL
LIN {X 0,Y 546.301,Z 691.44,A -85,B 0,C 180,E1 3797.948,E2 3797.948} C_VEL
LIN {X 0,Y 546.325,Z 691.44,A -85,B 0,C 180,E1 3801.514,E2 3801.514} C_VEL
LIN {X 0,Y 542.331,Z 691.44,A -85,B 0,C 180,E1 3803.303,E2 3803.303} C_VEL
LIN {X 0,Y 538.378,Z 691.44,A -85,B 0,C 180,E1 3805.118,E2 3805.118} C_VEL
LIN {X 0,Y 538.233,Z 691.44,A -85,B 0,C 180,E1 3810.421,E2 3810.421} C_VEL
LIN {X 0,Y 538.233,Z 691.44,A -85,B 0,C 180,E1 3816.209,E2 3816.209} C_VEL
LIN {X 0,Y 538.204,Z 691.44,A -85,B 0,C 180,E1 3822.465,E2 3822.465} C_VEL
LIN {X 0,Y 538.129,Z 691.44,A -85,B 0,C 180,E1 3827.526,E2 3827.526} C_VEL
LIN {X 0,Y 538.259,Z 691.995,A -85,B 0,C 180,E1 3831.234,E2 3831.234} C_VEL
LIN {X 0,Y 552.546,Z 720.217,A -85,B 0,C 180,E1 3832.866,E2 3832.866} C_VEL
LIN {X 0,Y 551.655,Z 763.443,A -85,B 0,C 180,E1 3833.734,E2 3833.734} C_VEL
LIN {X 0,Y 550.13,Z 803.424,A -85,B 0,C 180,E1 3835.135,E2 3835.135} C_VEL
LIN {X 0,Y 547.996,Z 843.749,A -85,B 0,C 180,E1 3837.234,E2 3837.234} C_VEL
LIN {X 0,Y 545.633,Z 881.015,A -85,B 0,C 180,E1 3839.886,E2 3839.886} C_VEL
LIN {X 0,Y 543.336,Z 916.858,A -85,B 0,C 180,E1 3843.243,E2 3843.243} C_VEL
LIN {X 0,Y 541.488,Z 947.389,A -85,B 0,C 180,E1 3846.955,E2 3846.955} C_VEL
LIN {X 0,Y 540.144,Z 972.999,A -85,B 0,C 180,E1 3850.983,E2 3850.983} C_VEL
LIN {X 0,Y 539.445,Z 992.246,A -85,B 0,C 180,E1 3854.953,E2 3854.953} C_VEL
LIN {X 0,Y 539.074,Z 1007.136,A -85,B 0,C 180,E1 3859.125,E2 3859.125} C_VEL
LIN {X 0,Y 538.937,Z 1017.479,A -85,B 0,C 180,E1 3863.548,E2 3863.548} C_VEL
LIN {X 0,Y 538.873,Z 1021.628,A -85,B 0,C 180,E1 3866.779,E2 3866.779} C_VEL
LIN {X 0,Y 538.853,Z 1023,A -85,B 0,C 180,E1 3870,E2 3870} C_VEL
LIN {X 0,Y 538.929,Z 1021.627,A -85,B 0,C 180,E1 3873.221,E2 3873.221} C_VEL
LIN {X 0,Y 539.042,Z 1015.916,A -85,B 0,C 180,E1 3877.262,E2 3877.262} C_VEL
LIN {X 0,Y 539.133,Z 1005.773,A -85,B 0,C 180,E1 3881.338,E2 3881.338} C_VEL
LIN {X 0,Y 539.58,Z 988.714,A -85,B 0,C 180,E1 3885.878,E2 3885.878} C_VEL
LIN {X 0,Y 540.519,Z 965.966,A -85,B 0,C 180,E1 3890.237,E2 3890.237} C_VEL
LIN {X 0,Y 542.068,Z 937.673,A -85,B 0,C 180,E1 3894.33,E2 3894.33} C_VEL
LIN {X 0,Y 544.048,Z 906.153,A -85,B 0,C 180,E1 3897.857,E2 3897.857} C_VEL
LIN {X 0,Y 546.444,Z 869.086,A -85,B 0,C 180,E1 3901.045,E2 3901.045} C_VEL
LIN {X 0,Y 548.76,Z 830.183,A -85,B 0,C 180,E1 3903.555,E2 3903.555} C_VEL
LIN {X 0,Y 550.839,Z 788.698,A -85,B 0,C 180,E1 3905.453,E2 3905.453} C_VEL
LIN {X 0,Y 552.169,Z 751.897,A -85,B 0,C 180,E1 3906.542,E2 3906.542} C_VEL
LIN {X 0,Y 552.118,Z 719.37,A -85,B 0,C 180,E1 3907.181,E2 3907.181} C_VEL
LIN {X 0,Y 538.25,Z 692.126,A -85,B 0,C 180,E1 3908.764,E2 3908.764} C_VEL
LIN {X 0,Y 538.184,Z 691.44,A -85,B 0,C 180,E1 3914.695,E2 3914.695} C_VEL
LIN {X 0,Y 538.226,Z 691.44,A -85,B 0,C 180,E1 3919.685,E2 3919.685} C_VEL
LIN {X 0,Y 538.198,Z 691.44,A -85,B 0,C 180,E1 3925.762,E2 3925.762} C_VEL
LIN {X 0,Y 538.251,Z 691.44,A -85,B 0,C 180,E1 3931.432,E2 3931.432} C_VEL
LIN {X 0,Y 538.382,Z 691.44,A -85,B 0,C 180,E1 3936.813,E2 3936.813} C_VEL
LIN {X 0,Y 538.538,Z 691.44,A -85,B 0,C 180,E1 3941.984,E2 3941.984} C_VEL
LIN {X 0,Y 538.461,Z 691.44,A -85,B 0,C 180,E1 3948.646,E2 3948.646} C_VEL
LIN {X 0,Y 538.667,Z 691.44,A -85,B 0,C 180,E1 3955.16,E2 3955.16} C_VEL
LIN {X 0,Y 538.708,Z 691.44,A -85,B 0,C 180,E1 3959.996,E2 3959.996} C_VEL
LIN {X 0,Y 538.672,Z 691.44,A -85,B 0,C 180,E1 3964.833,E2 3964.833} C_VEL
LIN {X 0,Y 538.522,Z 691.44,A -85,B 0,C 180,E1 3970.248,E2 3970.248} C_VEL
LIN {X 0,Y 538.544,Z 691.44,A -85,B 0,C 180,E1 3974.651,E2 3974.651} C_VEL
LIN {X 0,Y 538.499,Z 691.44,A -85,B 0,C 180,E1 3979.712,E2 3979.712} C_VEL
LIN {X 0,Y 538.311,Z 691.44,A -85,B 0,C 180,E1 3985.835,E2 3985.835} C_VEL
LIN {X 0,Y 538.308,Z 691.44,A -85,B 0,C 180,E1 3990.407,E2 3990.407} C_VEL
LIN {X 0,Y 538.337,Z 691.44,A -85,B 0,C 180,E1 3996.191,E2 3996.191} C_VEL
LIN {X 0,Y 538.126,Z 691.44,A -85,B 0,C 180,E1 4002.462,E2 4002.462} C_VEL
LIN {X 0,Y 538.143,Z 691.44,A -85,B 0,C 180,E1 4007.526,E2 4007.526} C_VEL
LIN {X 0,Y 538.368,Z 691.44,A -85,B 0,C 180,E1 4011.68,E2 4011.68} C_VEL
LIN {X 0,Y 542.784,Z 701.28,A -85,B 0,C 180,E1 4012.225,E2 4012.225} C_VEL
LIN {X 0,Y 552.1,Z 721.429,A -85,B 0,C 180,E1 4013.396,E2 4013.396} C_VEL
LIN {X 0,Y 550.806,Z 759.697,A -85,B 0,C 180,E1 4014.543,E2 4014.543} C_VEL
LIN {X 0,Y 548.766,Z 799.911,A -85,B 0,C 180,E1 4016.385,E2 4016.385} C_VEL
LIN {X 0,Y 546.445,Z 838.35,A -85,B 0,C 180,E1 4018.854,E2 4018.854} C_VEL
LIN {X 0,Y 544.089,Z 874.686,A -85,B 0,C 180,E1 4021.955,E2 4021.955} C_VEL
LIN {X 0,Y 542.039,Z 908.032,A -85,B 0,C 180,E1 4025.668,E2 4025.668} C_VEL
LIN {X 0,Y 540.485,Z 936.177,A -85,B 0,C 180,E1 4029.752,E2 4029.752} C_VEL
LIN {X 0,Y 539.557,Z 958.915,A -85,B 0,C 180,E1 4034.121,E2 4034.121} C_VEL
LIN {X 0,Y 539.11,Z 975.92,A -85,B 0,C 180,E1 4038.662,E2 4038.662} C_VEL
LIN {X 0,Y 539.019,Z 986.003,A -85,B 0,C 180,E1 4042.738,E2 4042.738} C_VEL
LIN {X 0,Y 538.972,Z 991.665,A -85,B 0,C 180,E1 4046.779,E2 4046.779} C_VEL
LIN {X 0,Y 538.919,Z 992.633,A -85,B 0,C 180,E1 4051.61,E2 4051.61} C_VEL
LIN {X 0,Y 538.966,Z 988.636,A -85,B 0,C 180,E1 4055.642,E2 4055.642} C_VEL
LIN {X 0,Y 539.111,Z 980.313,A -85,B 0,C 180,E1 4059.701,E2 4059.701} C_VEL
LIN {X 0,Y 539.374,Z 965.561,A -85,B 0,C 180,E1 4064.204,E2 4064.204} C_VEL
LIN {X 0,Y 540.136,Z 945.067,A -85,B 0,C 180,E1 4068.594,E2 4068.594} C_VEL
LIN {X 0,Y 541.39,Z 918.958,A -85,B 0,C 180,E1 4072.782,E2 4072.782} C_VEL
LIN {X 0,Y 543.306,Z 887.584,A -85,B 0,C 180,E1 4076.636,E2 4076.636} C_VEL
LIN {X 0,Y 545.604,Z 852.256,A -85,B 0,C 180,E1 4079.967,E2 4079.967} C_VEL
LIN {X 0,Y 547.968,Z 814.286,A -85,B 0,C 180,E1 4082.689,E2 4082.689} C_VEL
LIN {X 0,Y 550.109,Z 774.178,A -85,B 0,C 180,E1 4084.784,E2 4084.784} C_VEL
LIN {X 0,Y 551.742,Z 734.19,A -85,B 0,C 180,E1 4086.192,E2 4086.192} C_VEL
LIN {X 0,Y 551.586,Z 719.214,A -85,B 0,C 180,E1 4086.609,E2 4086.609} C_VEL
LIN {X 0,Y 538.358,Z 693.082,A -85,B 0,C 180,E1 4088.193,E2 4088.193} C_VEL
LIN {X 0,Y 538.173,Z 691.44,A -85,B 0,C 180,E1 4088.239,E2 4088.239} C_VEL
LIN {X 0,Y 538.186,Z 691.44,A -85,B 0,C 180,E1 4094.694,E2 4094.694} C_VEL
LIN {X 0,Y 538.208,Z 691.44,A -85,B 0,C 180,E1 4099.693,E2 4099.693} C_VEL
LIN {X 0,Y 538.16,Z 691.44,A -85,B 0,C 180,E1 4105.768,E2 4105.768} C_VEL
LIN {X 0,Y 538.263,Z 691.44,A -85,B 0,C 180,E1 4111.441,E2 4111.441} C_VEL
LIN {X 0,Y 538.405,Z 691.44,A -85,B 0,C 180,E1 4116.823,E2 4116.823} C_VEL
LIN {X 0,Y 538.515,Z 691.44,A -85,B 0,C 180,E1 4121.991,E2 4121.991} C_VEL
LIN {X 0,Y 538.65,Z 691.44,A -85,B 0,C 180,E1 4127.011,E2 4127.011} C_VEL
LIN {X 0,Y 538.621,Z 691.44,A -85,B 0,C 180,E1 4131.925,E2 4131.925} C_VEL
LIN {X 0,Y 538.771,Z 691.44,A -85,B 0,C 180,E1 4136.782,E2 4136.782} C_VEL
LIN {X 0,Y 538.893,Z 691.44,A -85,B 0,C 180,E1 4141.614,E2 4141.614} C_VEL
LIN {X 0,Y 538.732,Z 691.44,A -85,B 0,C 180,E1 4146.458,E2 4146.458} C_VEL
LIN {X 0,Y 538.491,Z 691.44,A -85,B 0,C 180,E1 4153.001,E2 4153.001} C_VEL
LIN {X 0,Y 538.424,Z 691.44,A -85,B 0,C 180,E1 4158.02,E2 4158.02} C_VEL
LIN {X 0,Y 538.4,Z 691.44,A -85,B 0,C 180,E1 4163.186,E2 4163.186} C_VEL
LIN {X 0,Y 538.378,Z 691.44,A -85,B 0,C 180,E1 4165.118,E2 4165.118} C_VEL
LIN {X 0,Y 537.063,Z 691.44,A -85,B 0,C 180,E1 4166.041,E2 4166.041} C_VEL
LIN {X 0,Y 530.394,Z 691.44,A -85,B 0,C 180,E1 4168.551,E2 4168.551} C_VEL
LIN {X 0,Y 530.312,Z 691.44,A -85,B 0,C 180,E1 4168.789,E2 4168.789} C_VEL
LIN {X 0,Y 530.282,Z 691.44,A -85,B 0,C 180,E1 4174.823,E2 4174.823} C_VEL
LIN {X 0,Y 530.289,Z 691.44,A -85,B 0,C 180,E1 4181.047,E2 4181.047} C_VEL
LIN {X 0,Y 530.243,Z 691.44,A -85,B 0,C 180,E1 4186.741,E2 4186.741} C_VEL
LIN {X 0,Y 530.306,Z 691.44,A -85,B 0,C 180,E1 4190.522,E2 4190.522} C_VEL
LIN {X 0,Y 534.764,Z 701.362,A -85,B 0,C 180,E1 4191.091,E2 4191.091} C_VEL
LIN {X 0,Y 546.269,Z 724,A -85,B 0,C 180,E1 4192.428,E2 4192.428} C_VEL
LIN {X 0,Y 545.068,Z 767.827,A -85,B 0,C 180,E1 4193.362,E2 4193.362} C_VEL
LIN {X 0,Y 543.324,Z 807.414,A -85,B 0,C 180,E1 4194.834,E2 4194.834} C_VEL
LIN {X 0,Y 541,Z 846.607,A -85,B 0,C 180,E1 4196.952,E2 4196.952} C_VEL
LIN {X 0,Y 538.417,Z 883.863,A -85,B 0,C 180,E1 4199.686,E2 4199.686} C_VEL
LIN {X 0,Y 535.821,Z 919.341,A -85,B 0,C 180,E1 4203.121,E2 4203.121} C_VEL
LIN {X 0,Y 533.761,Z 950.21,A -85,B 0,C 180,E1 4207.015,E2 4207.015} C_VEL
LIN {X 0,Y 532.286,Z 975.303,A -85,B 0,C 180,E1 4211.122,E2 4211.122} C_VEL
LIN {X 0,Y 531.578,Z 993.987,A -85,B 0,C 180,E1 4215.147,E2 4215.147} C_VEL
LIN {X 0,Y 531.163,Z 1008.005,A -85,B 0,C 180,E1 4219.274,E2 4219.274} C_VEL
LIN {X 0,Y 531.062,Z 1017.479,A -85,B 0,C 180,E1 4223.452,E2 4223.452} C_VEL
LIN {X 0,Y 530.984,Z 1021.628,A -85,B 0,C 180,E1 4226.731,E2 4226.731} C_VEL
LIN {X 0,Y 530.953,Z 1023,A -85,B 0,C 180,E1 4230,E2 4230} C_VEL
LIN {X 0,Y 530.972,Z 1021.229,A -85,B 0,C 180,E1 4233.655,E2 4233.655} C_VEL
LIN {X 0,Y 531.103,Z 1014.33,A -85,B 0,C 180,E1 4238.195,E2 4238.195} C_VEL
LIN {X 0,Y 531.273,Z 1003.09,A -85,B 0,C 180,E1 4242.342,E2 4242.342} C_VEL
LIN {X 0,Y 531.836,Z 986.766,A -85,B 0,C 180,E1 4246.541,E2 4246.541} C_VEL
LIN {X 0,Y 532.951,Z 964.878,A -85,B 0,C 180,E1 4250.716,E2 4250.716} C_VEL
LIN {X 0,Y 534.619,Z 937.208,A -85,B 0,C 180,E1 4254.751,E2 4254.751} C_VEL
LIN {X 0,Y 536.825,Z 905.693,A -85,B 0,C 180,E1 4258.312,E2 4258.312} C_VEL
LIN {X 0,Y 539.405,Z 869.647,A -85,B 0,C 180,E1 4261.452,E2 4261.452} C_VEL
LIN {X 0,Y 542.039,Z 830.187,A -85,B 0,C 180,E1 4264.027,E2 4264.027} C_VEL
LIN {X 0,Y 544.328,Z 789.199,A -85,B 0,C 180,E1 4265.92,E2 4265.92} C_VEL
LIN {X 0,Y 545.83,Z 751.896,A -85,B 0,C 180,E1 4267.037,E2 4267.037} C_VEL
LIN {X 0,Y 545.955,Z 722.58,A -85,B 0,C 180,E1 4267.621,E2 4267.621} C_VEL
LIN {X 0,Y 530.363,Z 692.149,A -85,B 0,C 180,E1 4269.452,E2 4269.452} C_VEL
LIN {X 0,Y 530.28,Z 691.44,A -85,B 0,C 180,E1 4275.546,E2 4275.546} C_VEL
LIN {X 0,Y 530.299,Z 691.44,A -85,B 0,C 180,E1 4281.089,E2 4281.089} C_VEL
LIN {X 0,Y 530.261,Z 691.44,A -85,B 0,C 180,E1 4287.145,E2 4287.145} C_VEL
LIN {X 0,Y 530.373,Z 691.44,A -85,B 0,C 180,E1 4292.821,E2 4292.821} C_VEL
LIN {X 0,Y 530.518,Z 691.44,A -85,B 0,C 180,E1 4298.221,E2 4298.221} C_VEL
LIN {X 0,Y 530.54,Z 691.44,A -85,B 0,C 180,E1 4303.416,E2 4303.416} C_VEL
LIN {X 0,Y 530.58,Z 691.44,A -85,B 0,C 180,E1 4310.139,E2 4310.139} C_VEL
LIN {X 0,Y 530.761,Z 691.44,A -85,B 0,C 180,E1 4315.087,E2 4315.087} C_VEL
LIN {X 0,Y 530.808,Z 691.44,A -85,B 0,C 180,E1 4319.996,E2 4319.996} C_VEL
LIN {X 0,Y 530.759,Z 691.44,A -85,B 0,C 180,E1 4324.905,E2 4324.905} C_VEL
LIN {X 0,Y 530.673,Z 691.44,A -85,B 0,C 180,E1 4329.852,E2 4329.852} C_VEL
LIN {X 0,Y 530.625,Z 691.44,A -85,B 0,C 180,E1 4334.874,E2 4334.874} C_VEL
LIN {X 0,Y 530.552,Z 691.44,A -85,B 0,C 180,E1 4340.019,E2 4340.019} C_VEL
LIN {X 0,Y 530.436,Z 691.44,A -85,B 0,C 180,E1 4345.343,E2 4345.343} C_VEL
LIN {X 0,Y 530.35,Z 691.44,A -85,B 0,C 180,E1 4351.078,E2 4351.078} C_VEL
LIN {X 0,Y 530.354,Z 691.44,A -85,B 0,C 180,E1 4356.93,E2 4356.93} C_VEL
LIN {X 0,Y 530.175,Z 691.44,A -85,B 0,C 180,E1 4363.254,E2 4363.254} C_VEL
LIN {X 0,Y 530.267,Z 691.44,A -85,B 0,C 180,E1 4368.949,E2 4368.949} C_VEL
LIN {X 0,Y 530.452,Z 691.44,A -85,B 0,C 180,E1 4371.004,E2 4371.004} C_VEL
LIN {X 0,Y 534.874,Z 701.385,A -85,B 0,C 180,E1 4371.568,E2 4371.568} C_VEL
LIN {X 0,Y 545.671,Z 723.949,A -85,B 0,C 180,E1 4372.957,E2 4372.957} C_VEL
LIN {X 0,Y 544.212,Z 761.521,A -85,B 0,C 180,E1 4374.128,E2 4374.128} C_VEL
LIN {X 0,Y 541.99,Z 800.972,A -85,B 0,C 180,E1 4375.97,E2 4375.97} C_VEL
LIN {X 0,Y 539.356,Z 840.189,A -85,B 0,C 180,E1 4378.541,E2 4378.541} C_VEL
LIN {X 0,Y 536.632,Z 877.745,A -85,B 0,C 180,E1 4381.846,E2 4381.846} C_VEL
LIN {X 0,Y 534.437,Z 909.968,A -85,B 0,C 180,E1 4385.562,E2 4385.562} C_VEL
LIN {X 0,Y 532.739,Z 937.422,A -85,B 0,C 180,E1 4389.666,E2 4389.666} C_VEL
LIN {X 0,Y 531.752,Z 958.912,A -85,B 0,C 180,E1 4393.882,E2 4393.882} C_VEL
LIN {X 0,Y 531.227,Z 975.917,A -85,B 0,C 180,E1 4398.491,E2 4398.491} C_VEL
LIN {X 0,Y 531.108,Z 986.002,A -85,B 0,C 180,E1 4402.629,E2 4402.629} C_VEL
LIN {X 0,Y 531.064,Z 991.665,A -85,B 0,C 180,E1 4406.731,E2 4406.731} C_VEL
LIN {X 0,Y 531.014,Z 992.634,A -85,B 0,C 180,E1 4411.634,E2 4411.634} C_VEL
LIN {X 0,Y 531.061,Z 988.637,A -85,B 0,C 180,E1 4415.727,E2 4415.727} C_VEL
LIN {X 0,Y 531.233,Z 980.314,A -85,B 0,C 180,E1 4419.846,E2 4419.846} C_VEL
LIN {X 0,Y 531.557,Z 965.343,A -85,B 0,C 180,E1 4424.476,E2 4424.476} C_VEL
LIN {X 0,Y 532.378,Z 945.073,A -85,B 0,C 180,E1 4428.875,E2 4428.875} C_VEL
LIN {X 0,Y 533.845,Z 918.464,A -85,B 0,C 180,E1 4433.198,E2 4433.198} C_VEL
LIN {X 0,Y 536.027,Z 886.732,A -85,B 0,C 180,E1 4437.12,E2 4437.12} C_VEL
LIN {X 0,Y 538.503,Z 852.268,A -85,B 0,C 180,E1 4440.404,E2 4440.404} C_VEL
LIN {X 0,Y 541.146,Z 814.325,A -85,B 0,C 180,E1 4443.152,E2 4443.152} C_VEL
LIN {X 0,Y 543.495,Z 774.85,A -85,B 0,C 180,E1 4445.237,E2 4445.237} C_VEL
LIN {X 0,Y 545.27,Z 735.913,A -85,B 0,C 180,E1 4446.638,E2 4446.638} C_VEL
LIN {X 0,Y 545.186,Z 722.199,A -85,B 0,C 180,E1 4447.035,E2 4447.035} C_VEL
LIN {X 0,Y 530.329,Z 692.802,A -85,B 0,C 180,E1 4448.885,E2 4448.885} C_VEL
LIN {X 0,Y 530.182,Z 691.44,A -85,B 0,C 180,E1 4448.922,E2 4448.922} C_VEL
LIN {X 0,Y 530.259,Z 691.44,A -85,B 0,C 180,E1 4454.465,E2 4454.465} C_VEL
LIN {X 0,Y 530.277,Z 691.44,A -85,B 0,C 180,E1 4460.436,E2 4460.436} C_VEL
LIN {X 0,Y 530.258,Z 691.44,A -85,B 0,C 180,E1 4465.899,E2 4465.899} C_VEL
LIN {X 0,Y 530.353,Z 691.44,A -85,B 0,C 180,E1 4472.252,E2 4472.252} C_VEL
LIN {X 0,Y 530.541,Z 691.44,A -85,B 0,C 180,E1 4478.23,E2 4478.23} C_VEL
LIN {X 0,Y 530.633,Z 691.44,A -85,B 0,C 180,E1 4483.428,E2 4483.428} C_VEL
LIN {X 0,Y 530.659,Z 691.44,A -85,B 0,C 180,E1 4488.485,E2 4488.485} C_VEL
LIN {X 0,Y 530.683,Z 691.44,A -85,B 0,C 180,E1 4493.452,E2 4493.452} C_VEL
LIN {X 0,Y 530.736,Z 691.44,A -85,B 0,C 180,E1 4498.369,E2 4498.369} C_VEL
LIN {X 0,Y 530.729,Z 691.44,A -85,B 0,C 180,E1 4503.274,E2 4503.274} C_VEL
LIN {X 0,Y 530.61,Z 691.44,A -85,B 0,C 180,E1 4508.205,E2 4508.205} C_VEL
LIN {X 0,Y 530.531,Z 691.44,A -85,B 0,C 180,E1 4513.994,E2 4513.994} C_VEL
LIN {X 0,Y 530.509,Z 691.44,A -85,B 0,C 180,E1 4520.03,E2 4520.03} C_VEL
LIN {X 0,Y 530.491,Z 691.44,A -85,B 0,C 180,E1 4525.349,E2 4525.349} C_VEL
LIN {X 0,Y 530.312,Z 691.44,A -85,B 0,C 180,E1 4528.789,E2 4528.789} C_VEL
LIN {X 0,Y 527.774,Z 691.44,A -85,B 0,C 180,E1 4530.177,E2 4530.177} C_VEL
LIN {X 0,Y 522.396,Z 691.44,A -85,B 0,C 180,E1 4532.257,E2 4532.257} C_VEL
LIN {X 0,Y 522.321,Z 691.44,A -85,B 0,C 180,E1 4532.498,E2 4532.498} C_VEL
LIN {X 0,Y 522.349,Z 691.44,A -85,B 0,C 180,E1 4538.499,E2 4538.499} C_VEL
LIN {X 0,Y 522.409,Z 691.44,A -85,B 0,C 180,E1 4544.072,E2 4544.072} C_VEL
LIN {X 0,Y 522.354,Z 692.197,A -85,B 0,C 180,E1 4549.823,E2 4549.823} C_VEL
LIN {X 0,Y 539.862,Z 725.754,A -85,B 0,C 180,E1 4551.932,E2 4551.932} C_VEL
LIN {X 0,Y 538.629,Z 770.753,A -85,B 0,C 180,E1 4552.944,E2 4552.944} C_VEL
LIN {X 0,Y 536.531,Z 811.181,A -85,B 0,C 180,E1 4554.514,E2 4554.514} C_VEL
LIN {X 0,Y 533.963,Z 849.547,A -85,B 0,C 180,E1 4556.669,E2 4556.669} C_VEL
LIN {X 0,Y 531.299,Z 884.606,A -85,B 0,C 180,E1 4559.306,E2 4559.306} C_VEL
LIN {X 0,Y 528.501,Z 919.341,A -85,B 0,C 180,E1 4562.718,E2 4562.718} C_VEL
LIN {X 0,Y 526.31,Z 949.074,A -85,B 0,C 180,E1 4566.498,E2 4566.498} C_VEL
LIN {X 0,Y 524.67,Z 974.194,A -85,B 0,C 180,E1 4570.618,E2 4570.618} C_VEL
LIN {X 0,Y 523.75,Z 993.986,A -85,B 0,C 180,E1 4574.92,E2 4574.92} C_VEL
LIN {X 0,Y 523.291,Z 1007.868,A -85,B 0,C 180,E1 4579.06,E2 4579.06} C_VEL
LIN {X 0,Y 523.159,Z 1017.479,A -85,B 0,C 180,E1 4583.353,E2 4583.353} C_VEL
LIN {X 0,Y 523.103,Z 1021.628,A -85,B 0,C 180,E1 4586.682,E2 4586.682} C_VEL
LIN {X 0,Y 523.066,Z 1023,A -85,B 0,C 180,E1 4590,E2 4590} C_VEL
LIN {X 0,Y 523.134,Z 1021.627,A -85,B 0,C 180,E1 4593.319,E2 4593.319} C_VEL
LIN {X 0,Y 523.257,Z 1015.917,A -85,B 0,C 180,E1 4597.482,E2 4597.482} C_VEL
LIN {X 0,Y 523.373,Z 1005.772,A -85,B 0,C 180,E1 4601.684,E2 4601.684} C_VEL
LIN {X 0,Y 523.905,Z 990.488,A -85,B 0,C 180,E1 4605.936,E2 4605.936} C_VEL
LIN {X 0,Y 524.969,Z 969.375,A -85,B 0,C 180,E1 4610.249,E2 4610.249} C_VEL
LIN {X 0,Y 526.718,Z 943.276,A -85,B 0,C 180,E1 4614.309,E2 4614.309} C_VEL
LIN {X 0,Y 529.008,Z 913.192,A -85,B 0,C 180,E1 4617.948,E2 4617.948} C_VEL
LIN {X 0,Y 531.708,Z 879.122,A -85,B 0,C 180,E1 4621.153,E2 4621.153} C_VEL
LIN {X 0,Y 534.525,Z 841.988,A -85,B 0,C 180,E1 4623.815,E2 4623.815} C_VEL
LIN {X 0,Y 537.157,Z 802.39,A -85,B 0,C 180,E1 4625.885,E2 4625.885} C_VEL
LIN {X 0,Y 539.076,Z 761.449,A -85,B 0,C 180,E1 4627.317,E2 4627.317} C_VEL
LIN {X 0,Y 539.516,Z 725.063,A -85,B 0,C 180,E1 4628.109,E2 4628.109} C_VEL
LIN {X 0,Y 522.36,Z 692.141,A -85,B 0,C 180,E1 4630.177,E2 4630.177} C_VEL
LIN {X 0,Y 522.399,Z 691.44,A -85,B 0,C 180,E1 4636.435,E2 4636.435} C_VEL
LIN {X 0,Y 522.35,Z 691.44,A -85,B 0,C 180,E1 4642.505,E2 4642.505} C_VEL
LIN {X 0,Y 522.331,Z 691.44,A -85,B 0,C 180,E1 4648.549,E2 4648.549} C_VEL
LIN {X 0,Y 522.494,Z 691.44,A -85,B 0,C 180,E1 4654.235,E2 4654.235} C_VEL
LIN {X 0,Y 522.617,Z 691.44,A -85,B 0,C 180,E1 4659.655,E2 4659.655} C_VEL
LIN {X 0,Y 522.449,Z 691.44,A -85,B 0,C 180,E1 4664.879,E2 4664.879} C_VEL
LIN {X 0,Y 522.664,Z 691.44,A -85,B 0,C 180,E1 4670.043,E2 4670.043} C_VEL
LIN {X 0,Y 522.855,Z 691.44,A -85,B 0,C 180,E1 4675.013,E2 4675.013} C_VEL
LIN {X 0,Y 522.907,Z 691.44,A -85,B 0,C 180,E1 4679.996,E2 4679.996} C_VEL
LIN {X 0,Y 522.846,Z 691.44,A -85,B 0,C 180,E1 4684.979,E2 4684.979} C_VEL
LIN {X 0,Y 522.767,Z 691.44,A -85,B 0,C 180,E1 4690.021,E2 4690.021} C_VEL
LIN {X 0,Y 522.69,Z 691.44,A -85,B 0,C 180,E1 4695.106,E2 4695.106} C_VEL
LIN {X 0,Y 522.611,Z 691.44,A -85,B 0,C 180,E1 4700.337,E2 4700.337} C_VEL
LIN {X 0,Y 522.452,Z 691.44,A -85,B 0,C 180,E1 4706.052,E2 4706.052} C_VEL
